LIN {X 0,Y 523.95,Z 318.842,A -85,B 0,C 180,E1 -4818.689,E2 -4818.689} C_VEL
LIN {X 0,Y 523.908,Z 318.846,A -85,B 0,C 180,E1 -4821.08,E2 -4821.08} C_VEL
LIN {X 0,Y 523.913,Z 318.849,A -85,B 0,C 180,E1 -4823.826,E2 -4823.826} C_VEL
LIN {X 0,Y 523.931,Z 318.844,A -85,B 0,C 180,E1 -4826.635,E2 -4826.635} C_VEL
LIN {X 0,Y 523.944,Z 318.837,A -85,B 0,C 180,E1 -4829.355,E2 -4829.355} C_VEL
LIN {X 0,Y 523.929,Z 318.846,A -85,B 0,C 180,E1 -4832.289,E2 -4832.289} C_VEL
LIN {X 0,Y 523.909,Z 318.846,A -85,B 0,C 180,E1 -4835.427,E2 -4835.427} C_VEL
LIN {X 0,Y 523.932,Z 318.841,A -85,B 0,C 180,E1 -4838.766,E2 -4838.766} C_VEL
LIN {X 0,Y 523.923,Z 318.845,A -85,B 0,C 180,E1 -4841.22,E2 -4841.22} C_VEL
LIN {X 0,Y 523.907,Z 318.851,A -85,B 0,C 180,E1 -4843.638,E2 -4843.638} C_VEL
LIN {X 0,Y 523.909,Z 318.849,A -85,B 0,C 180,E1 -4846.027,E2 -4846.027} C_VEL
LIN {X 0,Y 523.947,Z 318.838,A -85,B 0,C 180,E1 -4848.393,E2 -4848.393} C_VEL
LIN {X 0,Y 523.93,Z 318.85,A -85,B 0,C 180,E1 -4851.515,E2 -4851.515} C_VEL
LIN {X 0,Y 524.049,Z 318.827,A -85,B 0,C 180,E1 -4854.614,E2 -4854.614} C_VEL
LIN {X 0,Y 524.086,Z 318.826,A -85,B 0,C 180,E1 -4857.695,E2 -4857.695} C_VEL
LIN {X 0,Y 524.076,Z 318.826,A -85,B 0,C 180,E1 -4860,E2 -4860} C_VEL
LIN {X 0,Y 524.024,Z 318.834,A -85,B 0,C 180,E1 -4863.075,E2 -4863.075} C_VEL
LIN {X 0,Y 524.002,Z 318.833,A -85,B 0,C 180,E1 -4866.16,E2 -4866.16} C_VEL
LIN {X 0,Y 523.966,Z 318.846,A -85,B 0,C 180,E1 -4869.263,E2 -4869.263} C_VEL
LIN {X 0,Y 523.984,Z 318.834,A -85,B 0,C 180,E1 -4871.736,E2 -4871.736} C_VEL
LIN {X 0,Y 523.979,Z 318.844,A -85,B 0,C 180,E1 -4875.052,E2 -4875.052} C_VEL
LIN {X 0,Y 523.935,Z 318.841,A -85,B 0,C 180,E1 -4877.97,E2 -4877.97} C_VEL
LIN {X 0,Y 523.96,Z 318.839,A -85,B 0,C 180,E1 -4880.411,E2 -4880.411} C_VEL
LIN {X 0,Y 523.9,Z 318.855,A -85,B 0,C 180,E1 -4882.894,E2 -4882.894} C_VEL
LIN {X 0,Y 523.942,Z 318.843,A -85,B 0,C 180,E1 -4885.42,E2 -4885.42} C_VEL
LIN {X 0,Y 523.956,Z 318.838,A -85,B 0,C 180,E1 -4888,E2 -4888} C_VEL
LIN {X 0,Y 523.936,Z 318.847,A -85,B 0,C 180,E1 -4890.856,E2 -4890.856} C_VEL
LIN {X 0,Y 523.953,Z 318.839,A -85,B 0,C 180,E1 -4893.736,E2 -4893.736} C_VEL
LIN {X 0,Y 523.897,Z 318.852,A -85,B 0,C 180,E1 -4896.402,E2 -4896.402} C_VEL
LIN {X 0,Y 523.917,Z 318.846,A -85,B 0,C 180,E1 -4899.086,E2 -4899.086} C_VEL
LIN {X 0,Y 523.948,Z 318.844,A -85,B 0,C 180,E1 -4902.12,E2 -4902.12} C_VEL
LIN {X 0,Y 523.95,Z 318.841,A -85,B 0,C 180,E1 -4905.31,E2 -4905.31} C_VEL
LIN {X 0,Y 523.912,Z 318.848,A -85,B 0,C 180,E1 -4906.88,E2 -4906.88} C_VEL
LIN {X 0,Y 523.238,Z 318.931,A -85,B 0,C 180,E1 -4907.522,E2 -4907.522} C_VEL
LIN {X 0,Y 520.371,Z 319.293,A -85,B 0,C 180,E1 -4908.563,E2 -4908.563} C_VEL
LIN {X 0,Y 517.964,Z 319.59,A -85,B 0,C 180,E1 -4909.402,E2 -4909.402} C_VEL
LIN {X 0,Y 516.952,Z 319.717,A -85,B 0,C 180,E1 -4910.05,E2 -4910.05} C_VEL
LIN {X 0,Y 516.88,Z 319.728,A -85,B 0,C 180,E1 -4910.269,E2 -4910.269} C_VEL
LIN {X 0,Y 516.883,Z 319.721,A -85,B 0,C 180,E1 -4913.343,E2 -4913.343} C_VEL
LIN {X 0,Y 516.912,Z 319.723,A -85,B 0,C 180,E1 -4916.122,E2 -4916.122} C_VEL
LIN {X 0,Y 516.892,Z 319.723,A -85,B 0,C 180,E1 -4918.937,E2 -4918.937} C_VEL
LIN {X 0,Y 516.979,Z 319.878,A -85,B 0,C 180,E1 -4921.229,E2 -4921.229} C_VEL
LIN {X 0,Y 518.392,Z 328.272,A -85,B 0,C 180,E1 -4922.771,E2 -4922.771} C_VEL
LIN {X 0,Y 517.957,Z 343.74,A -85,B 0,C 180,E1 -4925.421,E2 -4925.421} C_VEL
LIN {X 0,Y 520.45,Z 355.889,A -85,B 0,C 180,E1 -4925.7,E2 -4925.7} C_VEL
LIN {X 0,Y 519.688,Z 480.334,A -85,B 0,C 180,E1 -4927.462,E2 -4927.462} C_VEL
LIN {X 0,Y 519.494,Z 494.514,A -85,B 0,C 180,E1 -4927.82,E2 -4927.82} C_VEL
LIN {X 0,Y 519.162,Z 507.735,A -85,B 0,C 180,E1 -4928.301,E2 -4928.301} C_VEL
LIN {X 0,Y 518.827,Z 519.994,A -85,B 0,C 180,E1 -4928.891,E2 -4928.891} C_VEL
LIN {X 0,Y 518.403,Z 532.763,A -85,B 0,C 180,E1 -4929.672,E2 -4929.672} C_VEL
LIN {X 0,Y 517.994,Z 544.752,A -85,B 0,C 180,E1 -4930.586,E2 -4930.586} C_VEL
LIN {X 0,Y 517.618,Z 555.659,A -85,B 0,C 180,E1 -4931.599,E2 -4931.599} C_VEL
LIN {X 0,Y 517.261,Z 564.741,A -85,B 0,C 180,E1 -4932.608,E2 -4932.608} C_VEL
LIN {X 0,Y 516.954,Z 573.83,A -85,B 0,C 180,E1 -4933.818,E2 -4933.818} C_VEL
LIN {X 0,Y 516.721,Z 581.347,A -85,B 0,C 180,E1 -4935.024,E2 -4935.024} C_VEL
LIN {X 0,Y 516.572,Z 587.573,A -85,B 0,C 180,E1 -4936.227,E2 -4936.227} C_VEL
LIN {X 0,Y 516.394,Z 592.697,A -85,B 0,C 180,E1 -4937.423,E2 -4937.423} C_VEL
LIN {X 0,Y 516.349,Z 597.948,A -85,B 0,C 180,E1 -4939.015,E2 -4939.015} C_VEL
LIN {X 0,Y 516.193,Z 601.647,A -85,B 0,C 180,E1 -4940.597,E2 -4940.597} C_VEL
LIN {X 0,Y 516.229,Z 603.917,A -85,B 0,C 180,E1 -4942.176,E2 -4942.176} C_VEL
LIN {X 0,Y 516.297,Z 604.832,A -85,B 0,C 180,E1 -4943.748,E2 -4943.748} C_VEL
LIN {X 0,Y 516.214,Z 604.426,A -85,B 0,C 180,E1 -4945.315,E2 -4945.315} C_VEL
LIN {X 0,Y 516.273,Z 602.695,A -85,B 0,C 180,E1 -4946.879,E2 -4946.879} C_VEL
LIN {X 0,Y 516.21,Z 599.622,A -85,B 0,C 180,E1 -4948.44,E2 -4948.44} C_VEL
LIN {X 0,Y 516.286,Z 595.104,A -85,B 0,C 180,E1 -4950,E2 -4950} C_VEL
LIN {X 0,Y 516.389,Z 588.969,A -85,B 0,C 180,E1 -4951.56,E2 -4951.56} C_VEL
LIN {X 0,Y 516.674,Z 582.141,A -85,B 0,C 180,E1 -4952.924,E2 -4952.924} C_VEL
LIN {X 0,Y 516.926,Z 573.712,A -85,B 0,C 180,E1 -4954.288,E2 -4954.288} C_VEL
LIN {X 0,Y 517.277,Z 564.923,A -85,B 0,C 180,E1 -4955.457,E2 -4955.457} C_VEL
LIN {X 0,Y 517.665,Z 554.313,A -85,B 0,C 180,E1 -4956.626,E2 -4956.626} C_VEL
LIN {X 0,Y 518.044,Z 542.812,A -85,B 0,C 180,E1 -4957.667,E2 -4957.667} C_VEL
LIN {X 0,Y 518.539,Z 530.43,A -85,B 0,C 180,E1 -4958.574,E2 -4958.574} C_VEL
LIN {X 0,Y 518.93,Z 517.026,A -85,B 0,C 180,E1 -4959.353,E2 -4959.353} C_VEL
LIN {X 0,Y 519.286,Z 504.042,A -85,B 0,C 180,E1 -4959.936,E2 -4959.936} C_VEL
LIN {X 0,Y 519.641,Z 490.877,A -85,B 0,C 180,E1 -4960.372,E2 -4960.372} C_VEL
LIN {X 0,Y 519.764,Z 476.594,A -85,B 0,C 180,E1 -4960.69,E2 -4960.69} C_VEL
LIN {X 0,Y 520.359,Z 355.201,A -85,B 0,C 180,E1 -4962.402,E2 -4962.402} C_VEL
LIN {X 0,Y 517.922,Z 343.676,A -85,B 0,C 180,E1 -4962.676,E2 -4962.676} C_VEL
LIN {X 0,Y 518.392,Z 328.422,A -85,B 0,C 180,E1 -4965.286,E2 -4965.286} C_VEL
LIN {X 0,Y 517.492,Z 322.48,A -85,B 0,C 180,E1 -4966.367,E2 -4966.367} C_VEL
LIN {X 0,Y 516.924,Z 319.72,A -85,B 0,C 180,E1 -4966.894,E2 -4966.894} C_VEL
LIN {X 0,Y 516.936,Z 319.724,A -85,B 0,C 180,E1 -4969.869,E2 -4969.869} C_VEL
LIN {X 0,Y 516.87,Z 319.725,A -85,B 0,C 180,E1 -4972.389,E2 -4972.389} C_VEL
LIN {X 0,Y 516.878,Z 319.722,A -85,B 0,C 180,E1 -4974.929,E2 -4974.929} C_VEL
LIN {X 0,Y 516.929,Z 319.721,A -85,B 0,C 180,E1 -4977.532,E2 -4977.532} C_VEL
LIN {X 0,Y 516.893,Z 319.722,A -85,B 0,C 180,E1 -4980.203,E2 -4980.203} C_VEL
LIN {X 0,Y 516.897,Z 319.719,A -85,B 0,C 180,E1 -4982.946,E2 -4982.946} C_VEL
LIN {X 0,Y 516.888,Z 319.725,A -85,B 0,C 180,E1 -4985.778,E2 -4985.778} C_VEL
LIN {X 0,Y 516.88,Z 319.721,A -85,B 0,C 180,E1 -4988.715,E2 -4988.715} C_VEL
LIN {X 0,Y 516.908,Z 319.721,A -85,B 0,C 180,E1 -4991.774,E2 -4991.774} C_VEL
LIN {X 0,Y 516.919,Z 319.718,A -85,B 0,C 180,E1 -4995.009,E2 -4995.009} C_VEL
LIN {X 0,Y 516.908,Z 319.715,A -85,B 0,C 180,E1 -4998.398,E2 -4998.398} C_VEL
LIN {X 0,Y 516.874,Z 319.729,A -85,B 0,C 180,E1 -5001.283,E2 -5001.283} C_VEL
LIN {X 0,Y 516.865,Z 319.722,A -85,B 0,C 180,E1 -5004.219,E2 -5004.219} C_VEL
LIN {X 0,Y 516.873,Z 319.726,A -85,B 0,C 180,E1 -5007.051,E2 -5007.051} C_VEL
LIN {X 0,Y 516.882,Z 319.721,A -85,B 0,C 180,E1 -5009.795,E2 -5009.795} C_VEL
LIN {X 0,Y 516.914,Z 319.713,A -85,B 0,C 180,E1 -5012.466,E2 -5012.466} C_VEL
LIN {X 0,Y 516.845,Z 319.733,A -85,B 0,C 180,E1 -5015.068,E2 -5015.068} C_VEL
LIN {X 0,Y 516.858,Z 319.722,A -85,B 0,C 180,E1 -5017.621,E2 -5017.621} C_VEL
LIN {X 0,Y 516.917,Z 319.71,A -85,B 0,C 180,E1 -5020.129,E2 -5020.129} C_VEL
LIN {X 0,Y 516.883,Z 319.723,A -85,B 0,C 180,E1 -5022.594,E2 -5022.594} C_VEL
LIN {X 0,Y 516.927,Z 319.718,A -85,B 0,C 180,E1 -5025.029,E2 -5025.029} C_VEL
LIN {X 0,Y 516.953,Z 319.707,A -85,B 0,C 180,E1 -5028.233,E2 -5028.233} C_VEL
LIN {X 0,Y 516.937,Z 319.714,A -85,B 0,C 180,E1 -5031.399,E2 -5031.399} C_VEL
LIN {X 0,Y 516.969,Z 319.707,A -85,B 0,C 180,E1 -5033.756,E2 -5033.756} C_VEL
LIN {X 0,Y 516.964,Z 319.713,A -85,B 0,C 180,E1 -5036.882,E2 -5036.882} C_VEL
LIN {X 0,Y 516.95,Z 319.717,A -85,B 0,C 180,E1 -5038.442,E2 -5038.442} C_VEL
LIN {X 0,Y 517.075,Z 319.7,A -85,B 0,C 180,E1 -5040.779,E2 -5040.779} C_VEL
LIN {X 0,Y 516.927,Z 319.712,A -85,B 0,C 180,E1 -5043.117,E2 -5043.117} C_VEL
LIN {X 0,Y 516.955,Z 319.717,A -85,B 0,C 180,E1 -5046.244,E2 -5046.244} C_VEL
LIN {X 0,Y 516.918,Z 319.711,A -85,B 0,C 180,E1 -5049.39,E2 -5049.39} C_VEL
LIN {X 0,Y 516.938,Z 319.715,A -85,B 0,C 180,E1 -5051.807,E2 -5051.807} C_VEL
LIN {X 0,Y 516.931,Z 319.711,A -85,B 0,C 180,E1 -5055.146,E2 -5055.146} C_VEL
LIN {X 0,Y 516.898,Z 319.727,A -85,B 0,C 180,E1 -5058.223,E2 -5058.223} C_VEL
LIN {X 0,Y 516.892,Z 319.717,A -85,B 0,C 180,E1 -5060.702,E2 -5060.702} C_VEL
LIN {X 0,Y 516.877,Z 319.729,A -85,B 0,C 180,E1 -5064.074,E2 -5064.074} C_VEL
LIN {X 0,Y 516.884,Z 319.72,A -85,B 0,C 180,E1 -5066.66,E2 -5066.66} C_VEL
LIN {X 0,Y 516.898,Z 319.72,A -85,B 0,C 180,E1 -5069.524,E2 -5069.524} C_VEL
LIN {X 0,Y 516.885,Z 319.721,A -85,B 0,C 180,E1 -5072.544,E2 -5072.544} C_VEL
LIN {X 0,Y 516.866,Z 319.724,A -85,B 0,C 180,E1 -5075.332,E2 -5075.332} C_VEL
LIN {X 0,Y 516.871,Z 319.729,A -85,B 0,C 180,E1 -5077.944,E2 -5077.944} C_VEL
LIN {X 0,Y 516.876,Z 319.718,A -85,B 0,C 180,E1 -5080.742,E2 -5080.742} C_VEL
LIN {X 0,Y 516.875,Z 319.72,A -85,B 0,C 180,E1 -5082.832,E2 -5082.832} C_VEL
LIN {X 0,Y 516.916,Z 319.717,A -85,B 0,C 180,E1 -5085.011,E2 -5085.011} C_VEL
LIN {X 0,Y 516.909,Z 319.718,A -85,B 0,C 180,E1 -5088.399,E2 -5088.399} C_VEL
LIN {X 0,Y 516.875,Z 319.728,A -85,B 0,C 180,E1 -5091.285,E2 -5091.285} C_VEL
LIN {X 0,Y 516.884,Z 319.723,A -85,B 0,C 180,E1 -5094.222,E2 -5094.222} C_VEL
LIN {X 0,Y 516.892,Z 319.724,A -85,B 0,C 180,E1 -5097.054,E2 -5097.054} C_VEL
LIN {X 0,Y 516.889,Z 319.724,A -85,B 0,C 180,E1 -5099.797,E2 -5099.797} C_VEL
LIN {X 0,Y 516.924,Z 319.718,A -85,B 0,C 180,E1 -5102.468,E2 -5102.468} C_VEL
LIN {X 0,Y 516.958,Z 319.835,A -85,B 0,C 180,E1 -5103.831,E2 -5103.831} C_VEL
LIN {X 0,Y 519.186,Z 331.01,A -85,B 0,C 180,E1 -5105.616,E2 -5105.616} C_VEL
LIN {X 0,Y 518.581,Z 350.946,A -85,B 0,C 180,E1 -5108.537,E2 -5108.537} C_VEL
LIN {X 0,Y 517.999,Z 370.569,A -85,B 0,C 180,E1 -5111.367,E2 -5111.367} C_VEL
LIN {X 0,Y 520.414,Z 384.995,A -85,B 0,C 180,E1 -5111.669,E2 -5111.669} C_VEL
LIN {X 0,Y 519.633,Z 509.029,A -85,B 0,C 180,E1 -5113.424,E2 -5113.424} C_VEL
LIN {X 0,Y 519.37,Z 523.154,A -85,B 0,C 180,E1 -5113.781,E2 -5113.781} C_VEL
LIN {X 0,Y 519.054,Z 536.913,A -85,B 0,C 180,E1 -5114.289,E2 -5114.289} C_VEL
LIN {X 0,Y 518.638,Z 550.885,A -85,B 0,C 180,E1 -5114.98,E2 -5114.98} C_VEL
LIN {X 0,Y 518.213,Z 563.388,A -85,B 0,C 180,E1 -5115.771,E2 -5115.771} C_VEL
LIN {X 0,Y 517.75,Z 575.993,A -85,B 0,C 180,E1 -5116.758,E2 -5116.758} C_VEL
LIN {X 0,Y 517.401,Z 587.135,A -85,B 0,C 180,E1 -5117.836,E2 -5117.836} C_VEL
LIN {X 0,Y 517.093,Z 597.302,A -85,B 0,C 180,E1 -5119.031,E2 -5119.031} C_VEL
LIN {X 0,Y 516.779,Z 605.67,A -85,B 0,C 180,E1 -5120.213,E2 -5120.213} C_VEL
LIN {X 0,Y 516.582,Z 613.673,A -85,B 0,C 180,E1 -5121.59,E2 -5121.59} C_VEL
LIN {X 0,Y 516.401,Z 620.117,A -85,B 0,C 180,E1 -5122.965,E2 -5122.965} C_VEL
LIN {X 0,Y 516.407,Z 624.584,A -85,B 0,C 180,E1 -5124.142,E2 -5124.142} C_VEL
LIN {X 0,Y 516.264,Z 628.09,A -85,B 0,C 180,E1 -5125.315,E2 -5125.315} C_VEL
LIN {X 0,Y 516.324,Z 629.979,A -85,B 0,C 180,E1 -5126.098,E2 -5126.098} C_VEL
LIN {X 0,Y 516.259,Z 632.685,A -85,B 0,C 180,E1 -5127.659,E2 -5127.659} C_VEL
LIN {X 0,Y 516.157,Z 634.024,A -85,B 0,C 180,E1 -5129.22,E2 -5129.22} C_VEL
LIN {X 0,Y 516.157,Z 634.024,A -85,B 0,C 180,E1 -5130.78,E2 -5130.78} C_VEL
LIN {X 0,Y 516.259,Z 632.686,A -85,B 0,C 180,E1 -5132.341,E2 -5132.341} C_VEL
LIN {X 0,Y 516.324,Z 629.98,A -85,B 0,C 180,E1 -5133.902,E2 -5133.902} C_VEL
LIN {X 0,Y 516.367,Z 625.828,A -85,B 0,C 180,E1 -5135.467,E2 -5135.467} C_VEL
LIN {X 0,Y 516.401,Z 620.109,A -85,B 0,C 180,E1 -5137.035,E2 -5137.035} C_VEL
LIN {X 0,Y 516.582,Z 613.665,A -85,B 0,C 180,E1 -5138.41,E2 -5138.41} C_VEL
LIN {X 0,Y 516.778,Z 605.659,A -85,B 0,C 180,E1 -5139.787,E2 -5139.787} C_VEL
LIN {X 0,Y 517.078,Z 597.289,A -85,B 0,C 180,E1 -5140.969,E2 -5140.969} C_VEL
LIN {X 0,Y 517.413,Z 586.881,A -85,B 0,C 180,E1 -5142.19,E2 -5142.19} C_VEL
LIN {X 0,Y 517.782,Z 575.975,A -85,B 0,C 180,E1 -5143.241,E2 -5143.241} C_VEL
LIN {X 0,Y 518.21,Z 563.371,A -85,B 0,C 180,E1 -5144.229,E2 -5144.229} C_VEL
LIN {X 0,Y 518.658,Z 550.865,A -85,B 0,C 180,E1 -5145.019,E2 -5145.019} C_VEL
LIN {X 0,Y 519.055,Z 538.011,A -85,B 0,C 180,E1 -5145.661,E2 -5145.661} C_VEL
LIN {X 0,Y 519.318,Z 524.346,A -85,B 0,C 180,E1 -5146.18,E2 -5146.18} C_VEL
LIN {X 0,Y 519.612,Z 510.139,A -85,B 0,C 180,E1 -5146.551,E2 -5146.551} C_VEL
LIN {X 0,Y 519.846,Z 482.014,A -85,B 0,C 180,E1 -5146.973,E2 -5146.973} C_VEL
LIN {X 0,Y 520.349,Z 384.013,A -85,B 0,C 180,E1 -5148.347,E2 -5148.347} C_VEL
LIN {X 0,Y 518,Z 370.517,A -85,B 0,C 180,E1 -5148.636,E2 -5148.636} C_VEL
LIN {X 0,Y 518.599,Z 349.484,A -85,B 0,C 180,E1 -5151.671,E2 -5151.671} C_VEL
LIN {X 0,Y 519.182,Z 330.987,A -85,B 0,C 180,E1 -5154.384,E2 -5154.384} C_VEL
LIN {X 0,Y 516.941,Z 319.775,A -85,B 0,C 180,E1 -5156.195,E2 -5156.195} C_VEL
LIN {X 0,Y 516.919,Z 319.719,A -85,B 0,C 180,E1 -5159.304,E2 -5159.304} C_VEL
LIN {X 0,Y 516.892,Z 319.728,A -85,B 0,C 180,E1 -5162.543,E2 -5162.543} C_VEL
LIN {X 0,Y 516.875,Z 319.722,A -85,B 0,C 180,E1 -5165.331,E2 -5165.331} C_VEL
LIN {X 0,Y 516.876,Z 319.72,A -85,B 0,C 180,E1 -5167.942,E2 -5167.942} C_VEL
LIN {X 0,Y 516.878,Z 319.722,A -85,B 0,C 180,E1 -5170.741,E2 -5170.741} C_VEL
LIN {X 0,Y 516.876,Z 319.721,A -85,B 0,C 180,E1 -5172.831,E2 -5172.831} C_VEL
LIN {X 0,Y 516.916,Z 319.714,A -85,B 0,C 180,E1 -5175.009,E2 -5175.009} C_VEL
LIN {X 0,Y 516.907,Z 319.723,A -85,B 0,C 180,E1 -5178.398,E2 -5178.398} C_VEL
LIN {X 0,Y 516.871,Z 319.722,A -85,B 0,C 180,E1 -5181.283,E2 -5181.283} C_VEL
LIN {X 0,Y 516.876,Z 319.727,A -85,B 0,C 180,E1 -5184.22,E2 -5184.22} C_VEL
LIN {X 0,Y 516.884,Z 319.72,A -85,B 0,C 180,E1 -5187.052,E2 -5187.052} C_VEL
LIN {X 0,Y 516.88,Z 319.719,A -85,B 0,C 180,E1 -5189.796,E2 -5189.796} C_VEL
LIN {X 0,Y 516.881,Z 319.722,A -85,B 0,C 180,E1 -5192.465,E2 -5192.465} C_VEL
LIN {X 0,Y 516.853,Z 319.723,A -85,B 0,C 180,E1 -5195.069,E2 -5195.069} C_VEL
LIN {X 0,Y 516.856,Z 319.729,A -85,B 0,C 180,E1 -5197.621,E2 -5197.621} C_VEL
LIN {X 0,Y 516.916,Z 319.72,A -85,B 0,C 180,E1 -5200.129,E2 -5200.129} C_VEL
LIN {X 0,Y 516.881,Z 319.72,A -85,B 0,C 180,E1 -5202.595,E2 -5202.595} C_VEL
LIN {X 0,Y 516.921,Z 319.715,A -85,B 0,C 180,E1 -5205.03,E2 -5205.03} C_VEL
LIN {X 0,Y 516.911,Z 319.715,A -85,B 0,C 180,E1 -5208.233,E2 -5208.233} C_VEL
LIN {X 0,Y 516.904,Z 319.725,A -85,B 0,C 180,E1 -5211.399,E2 -5211.399} C_VEL
LIN {X 0,Y 516.995,Z 319.706,A -85,B 0,C 180,E1 -5214.54,E2 -5214.54} C_VEL
LIN {X 0,Y 517.058,Z 319.701,A -85,B 0,C 180,E1 -5217.663,E2 -5217.663} C_VEL
LIN {X 0,Y 517.045,Z 319.701,A -85,B 0,C 180,E1 -5220,E2 -5220} C_VEL
LIN {X 0,Y 517.059,Z 319.696,A -85,B 0,C 180,E1 -5222.337,E2 -5222.337} C_VEL
LIN {X 0,Y 517,Z 319.711,A -85,B 0,C 180,E1 -5225.461,E2 -5225.461} C_VEL
LIN {X 0,Y 516.948,Z 319.712,A -85,B 0,C 180,E1 -5227.814,E2 -5227.814} C_VEL
LIN {X 0,Y 516.931,Z 319.721,A -85,B 0,C 180,E1 -5230.973,E2 -5230.973} C_VEL
LIN {X 0,Y 516.872,Z 319.722,A -85,B 0,C 180,E1 -5234.167,E2 -5234.167} C_VEL
LIN {X 0,Y 516.894,Z 319.72,A -85,B 0,C 180,E1 -5236.591,E2 -5236.591} C_VEL
LIN {X 0,Y 516.888,Z 319.727,A -85,B 0,C 180,E1 -5239.046,E2 -5239.046} C_VEL
LIN {X 0,Y 516.874,Z 319.723,A -85,B 0,C 180,E1 -5241.539,E2 -5241.539} C_VEL
LIN {X 0,Y 516.898,Z 319.725,A -85,B 0,C 180,E1 -5244.929,E2 -5244.929} C_VEL
LIN {X 0,Y 516.913,Z 319.715,A -85,B 0,C 180,E1 -5247.906,E2 -5247.906} C_VEL
LIN {X 0,Y 516.883,Z 319.722,A -85,B 0,C 180,E1 -5250.205,E2 -5250.205} C_VEL
LIN {X 0,Y 516.889,Z 319.724,A -85,B 0,C 180,E1 -5252.948,E2 -5252.948} C_VEL
LIN {X 0,Y 516.865,Z 319.722,A -85,B 0,C 180,E1 -5255.781,E2 -5255.781} C_VEL
LIN {X 0,Y 516.876,Z 319.727,A -85,B 0,C 180,E1 -5258.717,E2 -5258.717} C_VEL
LIN {X 0,Y 516.909,Z 319.718,A -85,B 0,C 180,E1 -5261.776,E2 -5261.776} C_VEL
LIN {X 0,Y 516.919,Z 319.718,A -85,B 0,C 180,E1 -5265.011,E2 -5265.011} C_VEL
LIN {X 0,Y 516.912,Z 319.724,A -85,B 0,C 180,E1 -5268.4,E2 -5268.4} C_VEL
LIN {X 0,Y 516.88,Z 319.728,A -85,B 0,C 180,E1 -5270.269,E2 -5270.269} C_VEL
LIN {X 0,Y 516.244,Z 319.814,A -85,B 0,C 180,E1 -5270.919,E2 -5270.919} C_VEL
LIN {X 0,Y 513.402,Z 320.167,A -85,B 0,C 180,E1 -5271.974,E2 -5271.974} C_VEL
LIN {X 0,Y 510.975,Z 320.463,A -85,B 0,C 180,E1 -5272.824,E2 -5272.824} C_VEL
LIN {X 0,Y 509.921,Z 320.59,A -85,B 0,C 180,E1 -5273.481,E2 -5273.481} C_VEL
LIN {X 0,Y 509.831,Z 320.601,A -85,B 0,C 180,E1 -5273.703,E2 -5273.703} C_VEL
LIN {X 0,Y 509.862,Z 320.601,A -85,B 0,C 180,E1 -5276.54,E2 -5276.54} C_VEL
LIN {X 0,Y 509.847,Z 320.601,A -85,B 0,C 180,E1 -5279.335,E2 -5279.335} C_VEL
LIN {X 0,Y 509.901,Z 320.629,A -85,B 0,C 180,E1 -5280.989,E2 -5280.989} C_VEL
LIN {X 0,Y 511.449,Z 329.163,A -85,B 0,C 180,E1 -5282.592,E2 -5282.592} C_VEL
LIN {X 0,Y 511.05,Z 343.771,A -85,B 0,C 180,E1 -5285.132,E2 -5285.132} C_VEL
LIN {X 0,Y 511.206,Z 344.967,A -85,B 0,C 180,E1 -5285.193,E2 -5285.193} C_VEL
LIN {X 0,Y 513.725,Z 357.045,A -85,B 0,C 180,E1 -5285.465,E2 -5285.465} C_VEL
LIN {X 0,Y 512.908,Z 480.339,A -85,B 0,C 180,E1 -5287.233,E2 -5287.233} C_VEL
LIN {X 0,Y 512.696,Z 494.434,A -85,B 0,C 180,E1 -5287.589,E2 -5287.589} C_VEL
LIN {X 0,Y 512.328,Z 508.308,A -85,B 0,C 180,E1 -5288.103,E2 -5288.103} C_VEL
LIN {X 0,Y 511.96,Z 520.665,A -85,B 0,C 180,E1 -5288.71,E2 -5288.71} C_VEL
LIN {X 0,Y 511.514,Z 533.228,A -85,B 0,C 180,E1 -5289.494,E2 -5289.494} C_VEL
LIN {X 0,Y 511.065,Z 545.144,A -85,B 0,C 180,E1 -5290.416,E2 -5290.416} C_VEL
LIN {X 0,Y 510.718,Z 555.025,A -85,B 0,C 180,E1 -5291.341,E2 -5291.341} C_VEL
LIN {X 0,Y 510.313,Z 564.247,A -85,B 0,C 180,E1 -5292.364,E2 -5292.364} C_VEL
LIN {X 0,Y 509.937,Z 573.452,A -85,B 0,C 180,E1 -5293.589,E2 -5293.589} C_VEL
LIN {X 0,Y 509.679,Z 581.963,A -85,B 0,C 180,E1 -5294.973,E2 -5294.973} C_VEL
LIN {X 0,Y 509.446,Z 589.219,A -85,B 0,C 180,E1 -5296.437,E2 -5296.437} C_VEL
LIN {X 0,Y 509.314,Z 594.04,A -85,B 0,C 180,E1 -5297.65,E2 -5297.65} C_VEL
LIN {X 0,Y 509.226,Z 598.997,A -85,B 0,C 180,E1 -5299.262,E2 -5299.262} C_VEL
LIN {X 0,Y 509.108,Z 601.696,A -85,B 0,C 180,E1 -5300.465,E2 -5300.465} C_VEL
LIN {X 0,Y 509.143,Z 604.035,A -85,B 0,C 180,E1 -5302.066,E2 -5302.066} C_VEL
LIN {X 0,Y 509.223,Z 605.016,A -85,B 0,C 180,E1 -5303.661,E2 -5303.661} C_VEL
LIN {X 0,Y 509.13,Z 604.677,A -85,B 0,C 180,E1 -5305.249,E2 -5305.249} C_VEL
LIN {X 0,Y 509.189,Z 603.012,A -85,B 0,C 180,E1 -5306.835,E2 -5306.835} C_VEL
LIN {X 0,Y 509.129,Z 600.008,A -85,B 0,C 180,E1 -5308.418,E2 -5308.418} C_VEL
LIN {X 0,Y 509.203,Z 595.577,A -85,B 0,C 180,E1 -5310,E2 -5310} C_VEL
LIN {X 0,Y 509.359,Z 591.183,A -85,B 0,C 180,E1 -5311.186,E2 -5311.186} C_VEL
LIN {X 0,Y 509.402,Z 585.867,A -85,B 0,C 180,E1 -5312.372,E2 -5312.372} C_VEL
LIN {X 0,Y 509.809,Z 578.244,A -85,B 0,C 180,E1 -5313.754,E2 -5313.754} C_VEL
LIN {X 0,Y 510.036,Z 570.335,A -85,B 0,C 180,E1 -5314.94,E2 -5314.94} C_VEL
LIN {X 0,Y 510.472,Z 560.809,A -85,B 0,C 180,E1 -5316.125,E2 -5316.125} C_VEL
LIN {X 0,Y 510.846,Z 551.329,A -85,B 0,C 180,E1 -5317.112,E2 -5317.112} C_VEL
LIN {X 0,Y 511.261,Z 539.04,A -85,B 0,C 180,E1 -5318.169,E2 -5318.169} C_VEL
LIN {X 0,Y 511.764,Z 527.273,A -85,B 0,C 180,E1 -5318.987,E2 -5318.987} C_VEL
LIN {X 0,Y 512.184,Z 514.945,A -85,B 0,C 180,E1 -5319.676,E2 -5319.676} C_VEL
LIN {X 0,Y 512.523,Z 501.271,A -85,B 0,C 180,E1 -5320.268,E2 -5320.268} C_VEL
LIN {X 0,Y 512.864,Z 486.886,A -85,B 0,C 180,E1 -5320.711,E2 -5320.711} C_VEL
LIN {X 0,Y 513.026,Z 472.695,A -85,B 0,C 180,E1 -5320.982,E2 -5320.982} C_VEL
LIN {X 0,Y 513.669,Z 356.374,A -85,B 0,C 180,E1 -5322.636,E2 -5322.636} C_VEL
LIN {X 0,Y 511.017,Z 343.888,A -85,B 0,C 180,E1 -5322.934,E2 -5322.934} C_VEL
LIN {X 0,Y 511.469,Z 329.787,A -85,B 0,C 180,E1 -5325.376,E2 -5325.376} C_VEL
LIN {X 0,Y 510.169,Z 322.01,A -85,B 0,C 180,E1 -5326.815,E2 -5326.815} C_VEL
LIN {X 0,Y 509.898,Z 320.596,A -85,B 0,C 180,E1 -5327.082,E2 -5327.082} C_VEL
LIN {X 0,Y 509.89,Z 320.597,A -85,B 0,C 180,E1 -5330.401,E2 -5330.401} C_VEL
LIN {X 0,Y 509.825,Z 320.605,A -85,B 0,C 180,E1 -5333.563,E2 -5333.563} C_VEL
LIN {X 0,Y 509.914,Z 320.591,A -85,B 0,C 180,E1 -5336.378,E2 -5336.378} C_VEL
LIN {X 0,Y 509.877,Z 320.592,A -85,B 0,C 180,E1 -5338.843,E2 -5338.843} C_VEL
LIN {X 0,Y 509.823,Z 320.607,A -85,B 0,C 180,E1 -5341.589,E2 -5341.589} C_VEL
LIN {X 0,Y 509.853,Z 320.596,A -85,B 0,C 180,E1 -5344.412,E2 -5344.412} C_VEL
LIN {X 0,Y 509.817,Z 320.605,A -85,B 0,C 180,E1 -5347.339,E2 -5347.339} C_VEL
LIN {X 0,Y 509.835,Z 320.592,A -85,B 0,C 180,E1 -5350.381,E2 -5350.381} C_VEL
LIN {X 0,Y 509.819,Z 320.603,A -85,B 0,C 180,E1 -5353.061,E2 -5353.061} C_VEL
LIN {X 0,Y 509.827,Z 320.603,A -85,B 0,C 180,E1 -5355.791,E2 -5355.791} C_VEL
LIN {X 0,Y 509.85,Z 320.595,A -85,B 0,C 180,E1 -5358.573,E2 -5358.573} C_VEL
LIN {X 0,Y 509.844,Z 320.597,A -85,B 0,C 180,E1 -5361.785,E2 -5361.785} C_VEL
LIN {X 0,Y 509.824,Z 320.601,A -85,B 0,C 180,E1 -5364.621,E2 -5364.621} C_VEL
LIN {X 0,Y 509.851,Z 320.6,A -85,B 0,C 180,E1 -5367.48,E2 -5367.48} C_VEL
LIN {X 0,Y 509.85,Z 320.596,A -85,B 0,C 180,E1 -5370.273,E2 -5370.273} C_VEL
LIN {X 0,Y 509.865,Z 320.596,A -85,B 0,C 180,E1 -5372.943,E2 -5372.943} C_VEL
LIN {X 0,Y 509.83,Z 320.601,A -85,B 0,C 180,E1 -5375.572,E2 -5375.572} C_VEL
LIN {X 0,Y 509.81,Z 320.599,A -85,B 0,C 180,E1 -5378.148,E2 -5378.148} C_VEL
LIN {X 0,Y 509.845,Z 320.596,A -85,B 0,C 180,E1 -5380.68,E2 -5380.68} C_VEL
LIN {X 0,Y 509.852,Z 320.6,A -85,B 0,C 180,E1 -5383.173,E2 -5383.173} C_VEL
LIN {X 0,Y 509.843,Z 320.594,A -85,B 0,C 180,E1 -5385.633,E2 -5385.633} C_VEL
LIN {X 0,Y 509.894,Z 320.595,A -85,B 0,C 180,E1 -5388.874,E2 -5388.874} C_VEL
LIN {X 0,Y 509.906,Z 320.59,A -85,B 0,C 180,E1 -5392.077,E2 -5392.077} C_VEL
LIN {X 0,Y 509.949,Z 320.587,A -85,B 0,C 180,E1 -5394.464,E2 -5394.464} C_VEL
LIN {X 0,Y 510.028,Z 320.572,A -85,B 0,C 180,E1 -5397.631,E2 -5397.631} C_VEL
LIN {X 0,Y 510.024,Z 320.578,A -85,B 0,C 180,E1 -5400.789,E2 -5400.789} C_VEL
LIN {X 0,Y 509.871,Z 320.591,A -85,B 0,C 180,E1 -5403.16,E2 -5403.16} C_VEL
LIN {X 0,Y 509.903,Z 320.597,A -85,B 0,C 180,E1 -5406.33,E2 -5406.33} C_VEL
LIN {X 0,Y 509.858,Z 320.591,A -85,B 0,C 180,E1 -5409.521,E2 -5409.521} C_VEL
LIN {X 0,Y 509.89,Z 320.594,A -85,B 0,C 180,E1 -5411.932,E2 -5411.932} C_VEL
LIN {X 0,Y 509.881,Z 320.589,A -85,B 0,C 180,E1 -5415.242,E2 -5415.242} C_VEL
LIN {X 0,Y 509.843,Z 320.601,A -85,B 0,C 180,E1 -5418.484,E2 -5418.484} C_VEL
LIN {X 0,Y 509.833,Z 320.594,A -85,B 0,C 180,E1 -5421.002,E2 -5421.002} C_VEL
LIN {X 0,Y 509.809,Z 320.602,A -85,B 0,C 180,E1 -5423.564,E2 -5423.564} C_VEL
LIN {X 0,Y 509.866,Z 320.597,A -85,B 0,C 180,E1 -5426.371,E2 -5426.371} C_VEL
LIN {X 0,Y 509.846,Z 320.602,A -85,B 0,C 180,E1 -5429.752,E2 -5429.752} C_VEL
LIN {X 0,Y 509.862,Z 320.595,A -85,B 0,C 180,E1 -5432.775,E2 -5432.775} C_VEL
LIN {X 0,Y 509.827,Z 320.603,A -85,B 0,C 180,E1 -5435.581,E2 -5435.581} C_VEL
LIN {X 0,Y 509.84,Z 320.6,A -85,B 0,C 180,E1 -5438.339,E2 -5438.339} C_VEL
LIN {X 0,Y 509.849,Z 320.598,A -85,B 0,C 180,E1 -5441.426,E2 -5441.426} C_VEL
LIN {X 0,Y 509.85,Z 320.596,A -85,B 0,C 180,E1 -5444.669,E2 -5444.669} C_VEL
LIN {X 0,Y 509.851,Z 320.599,A -85,B 0,C 180,E1 -5448.104,E2 -5448.104} C_VEL
LIN {X 0,Y 509.84,Z 320.599,A -85,B 0,C 180,E1 -5450.648,E2 -5450.648} C_VEL
LIN {X 0,Y 509.83,Z 320.608,A -85,B 0,C 180,E1 -5453.649,E2 -5453.649} C_VEL
LIN {X 0,Y 509.857,Z 320.597,A -85,B 0,C 180,E1 -5456.54,E2 -5456.54} C_VEL
LIN {X 0,Y 509.842,Z 320.605,A -85,B 0,C 180,E1 -5459.335,E2 -5459.335} C_VEL
LIN {X 0,Y 509.89,Z 320.596,A -85,B 0,C 180,E1 -5462.055,E2 -5462.055} C_VEL
LIN {X 0,Y 509.914,Z 320.746,A -85,B 0,C 180,E1 -5463.621,E2 -5463.621} C_VEL
LIN {X 0,Y 512.29,Z 332.48,A -85,B 0,C 180,E1 -5465.521,E2 -5465.521} C_VEL
LIN {X 0,Y 511.646,Z 352.18,A -85,B 0,C 180,E1 -5468.443,E2 -5468.443} C_VEL
LIN {X 0,Y 511.076,Z 370.394,A -85,B 0,C 180,E1 -5471.109,E2 -5471.109} C_VEL
LIN {X 0,Y 513.687,Z 385.81,A -85,B 0,C 180,E1 -5471.435,E2 -5471.435} C_VEL
LIN {X 0,Y 512.817,Z 508.816,A -85,B 0,C 180,E1 -5473.197,E2 -5473.197} C_VEL
LIN {X 0,Y 512.527,Z 523.27,A -85,B 0,C 180,E1 -5473.569,E2 -5473.569} C_VEL
LIN {X 0,Y 512.206,Z 536.706,A -85,B 0,C 180,E1 -5474.073,E2 -5474.073} C_VEL
LIN {X 0,Y 511.771,Z 550.68,A -85,B 0,C 180,E1 -5474.774,E2 -5474.774} C_VEL
LIN {X 0,Y 511.273,Z 563.183,A -85,B 0,C 180,E1 -5475.573,E2 -5475.573} C_VEL
LIN {X 0,Y 510.805,Z 575.789,A -85,B 0,C 180,E1 -5476.575,E2 -5476.575} C_VEL
LIN {X 0,Y 510.409,Z 586.355,A -85,B 0,C 180,E1 -5477.604,E2 -5477.604} C_VEL
LIN {X 0,Y 510.063,Z 597.098,A -85,B 0,C 180,E1 -5478.878,E2 -5478.878} C_VEL
LIN {X 0,Y 509.732,Z 605.467,A -85,B 0,C 180,E1 -5480.076,E2 -5480.076} C_VEL
LIN {X 0,Y 509.522,Z 613.471,A -85,B 0,C 180,E1 -5481.473,E2 -5481.473} C_VEL
LIN {X 0,Y 509.326,Z 619.915,A -85,B 0,C 180,E1 -5482.866,E2 -5482.866} C_VEL
LIN {X 0,Y 509.304,Z 624.382,A -85,B 0,C 180,E1 -5484.06,E2 -5484.06} C_VEL
LIN {X 0,Y 509.181,Z 627.889,A -85,B 0,C 180,E1 -5485.25,E2 -5485.25} C_VEL
LIN {X 0,Y 509.193,Z 631.305,A -85,B 0,C 180,E1 -5486.835,E2 -5486.835} C_VEL
LIN {X 0,Y 509.109,Z 633.322,A -85,B 0,C 180,E1 -5488.418,E2 -5488.418} C_VEL
LIN {X 0,Y 509.064,Z 633.99,A -85,B 0,C 180,E1 -5490,E2 -5490} C_VEL
LIN {X 0,Y 509.109,Z 633.322,A -85,B 0,C 180,E1 -5491.582,E2 -5491.582} C_VEL
LIN {X 0,Y 509.193,Z 631.305,A -85,B 0,C 180,E1 -5493.165,E2 -5493.165} C_VEL
LIN {X 0,Y 509.181,Z 627.886,A -85,B 0,C 180,E1 -5494.75,E2 -5494.75} C_VEL
LIN {X 0,Y 509.303,Z 624.373,A -85,B 0,C 180,E1 -5495.94,E2 -5495.94} C_VEL
LIN {X 0,Y 509.326,Z 619.904,A -85,B 0,C 180,E1 -5497.134,E2 -5497.134} C_VEL
LIN {X 0,Y 509.522,Z 613.46,A -85,B 0,C 180,E1 -5498.527,E2 -5498.527} C_VEL
LIN {X 0,Y 509.731,Z 605.452,A -85,B 0,C 180,E1 -5499.924,E2 -5499.924} C_VEL
LIN {X 0,Y 510.047,Z 597.081,A -85,B 0,C 180,E1 -5501.122,E2 -5501.122} C_VEL
LIN {X 0,Y 510.411,Z 586.364,A -85,B 0,C 180,E1 -5502.393,E2 -5502.393} C_VEL
LIN {X 0,Y 510.819,Z 575.765,A -85,B 0,C 180,E1 -5503.425,E2 -5503.425} C_VEL
LIN {X 0,Y 511.231,Z 564.59,A -85,B 0,C 180,E1 -5504.326,E2 -5504.326} C_VEL
LIN {X 0,Y 511.687,Z 552.424,A -85,B 0,C 180,E1 -5505.127,E2 -5505.127} C_VEL
LIN {X 0,Y 512.167,Z 538.93,A -85,B 0,C 180,E1 -5505.826,E2 -5505.826} C_VEL
LIN {X 0,Y 512.466,Z 524.772,A -85,B 0,C 180,E1 -5506.381,E2 -5506.381} C_VEL
LIN {X 0,Y 512.814,Z 509.919,A -85,B 0,C 180,E1 -5506.777,E2 -5506.777} C_VEL
LIN {X 0,Y 513.028,Z 483.59,A -85,B 0,C 180,E1 -5507.18,E2 -5507.18} C_VEL
LIN {X 0,Y 513.571,Z 384.829,A -85,B 0,C 180,E1 -5508.583,E2 -5508.583} C_VEL
LIN {X 0,Y 511.08,Z 370.329,A -85,B 0,C 180,E1 -5508.895,E2 -5508.895} C_VEL
LIN {X 0,Y 511.698,Z 349.298,A -85,B 0,C 180,E1 -5511.979,E2 -5511.979} C_VEL
LIN {X 0,Y 512.29,Z 332.536,A -85,B 0,C 180,E1 -5514.479,E2 -5514.479} C_VEL
LIN {X 0,Y 510.286,Z 322.35,A -85,B 0,C 180,E1 -5516.149,E2 -5516.149} C_VEL
LIN {X 0,Y 509.905,Z 320.598,A -85,B 0,C 180,E1 -5516.485,E2 -5516.485} C_VEL
LIN {X 0,Y 509.874,Z 320.6,A -85,B 0,C 180,E1 -5518.844,E2 -5518.844} C_VEL
LIN {X 0,Y 509.816,Z 320.603,A -85,B 0,C 180,E1 -5521.589,E2 -5521.589} C_VEL
LIN {X 0,Y 509.848,Z 320.604,A -85,B 0,C 180,E1 -5524.413,E2 -5524.413} C_VEL
LIN {X 0,Y 509.814,Z 320.597,A -85,B 0,C 180,E1 -5527.34,E2 -5527.34} C_VEL
LIN {X 0,Y 509.832,Z 320.6,A -85,B 0,C 180,E1 -5530.381,E2 -5530.381} C_VEL
LIN {X 0,Y 509.816,Z 320.599,A -85,B 0,C 180,E1 -5533.061,E2 -5533.061} C_VEL
LIN {X 0,Y 509.823,Z 320.599,A -85,B 0,C 180,E1 -5535.792,E2 -5535.792} C_VEL
LIN {X 0,Y 509.849,Z 320.6,A -85,B 0,C 180,E1 -5538.574,E2 -5538.574} C_VEL
LIN {X 0,Y 509.842,Z 320.602,A -85,B 0,C 180,E1 -5541.786,E2 -5541.786} C_VEL
LIN {X 0,Y 509.83,Z 320.599,A -85,B 0,C 180,E1 -5544.622,E2 -5544.622} C_VEL
LIN {X 0,Y 509.851,Z 320.598,A -85,B 0,C 180,E1 -5547.48,E2 -5547.48} C_VEL
LIN {X 0,Y 509.847,Z 320.594,A -85,B 0,C 180,E1 -5550.273,E2 -5550.273} C_VEL
LIN {X 0,Y 509.863,Z 320.599,A -85,B 0,C 180,E1 -5553.629,E2 -5553.629} C_VEL
LIN {X 0,Y 509.809,Z 320.603,A -85,B 0,C 180,E1 -5556.436,E2 -5556.436} C_VEL
LIN {X 0,Y 509.903,Z 320.595,A -85,B 0,C 180,E1 -5559.844,E2 -5559.844} C_VEL
LIN {X 0,Y 509.85,Z 320.598,A -85,B 0,C 180,E1 -5563.174,E2 -5563.174} C_VEL
LIN {X 0,Y 509.838,Z 320.605,A -85,B 0,C 180,E1 -5565.634,E2 -5565.634} C_VEL
LIN {X 0,Y 509.875,Z 320.592,A -85,B 0,C 180,E1 -5568.131,E2 -5568.131} C_VEL
LIN {X 0,Y 509.857,Z 320.601,A -85,B 0,C 180,E1 -5571.279,E2 -5571.279} C_VEL
LIN {X 0,Y 509.946,Z 320.584,A -85,B 0,C 180,E1 -5574.464,E2 -5574.464} C_VEL
LIN {X 0,Y 510.028,Z 320.577,A -85,B 0,C 180,E1 -5577.631,E2 -5577.631} C_VEL
LIN {X 0,Y 510.015,Z 320.577,A -85,B 0,C 180,E1 -5580,E2 -5580} C_VEL
LIN {X 0,Y 510.03,Z 320.571,A -85,B 0,C 180,E1 -5582.369,E2 -5582.369} C_VEL
LIN {X 0,Y 509.952,Z 320.588,A -85,B 0,C 180,E1 -5585.536,E2 -5585.536} C_VEL
LIN {X 0,Y 509.907,Z 320.588,A -85,B 0,C 180,E1 -5587.923,E2 -5587.923} C_VEL
LIN {X 0,Y 509.895,Z 320.597,A -85,B 0,C 180,E1 -5591.126,E2 -5591.126} C_VEL
LIN {X 0,Y 509.844,Z 320.598,A -85,B 0,C 180,E1 -5594.367,E2 -5594.367} C_VEL
LIN {X 0,Y 509.866,Z 320.595,A -85,B 0,C 180,E1 -5597.653,E2 -5597.653} C_VEL
LIN {X 0,Y 509.875,Z 320.594,A -85,B 0,C 180,E1 -5600.402,E2 -5600.402} C_VEL
LIN {X 0,Y 509.819,Z 320.6,A -85,B 0,C 180,E1 -5603.564,E2 -5603.564} C_VEL
LIN {X 0,Y 509.901,Z 320.593,A -85,B 0,C 180,E1 -5606.379,E2 -5606.379} C_VEL
LIN {X 0,Y 509.866,Z 320.602,A -85,B 0,C 180,E1 -5608.845,E2 -5608.845} C_VEL
LIN {X 0,Y 509.813,Z 320.599,A -85,B 0,C 180,E1 -5611.591,E2 -5611.591} C_VEL
LIN {X 0,Y 509.843,Z 320.602,A -85,B 0,C 180,E1 -5614.415,E2 -5614.415} C_VEL
LIN {X 0,Y 509.81,Z 320.6,A -85,B 0,C 180,E1 -5617.342,E2 -5617.342} C_VEL
LIN {X 0,Y 509.833,Z 320.604,A -85,B 0,C 180,E1 -5620.383,E2 -5620.383} C_VEL
LIN {X 0,Y 509.819,Z 320.603,A -85,B 0,C 180,E1 -5623.063,E2 -5623.063} C_VEL
LIN {X 0,Y 509.827,Z 320.601,A -85,B 0,C 180,E1 -5625.794,E2 -5625.794} C_VEL
LIN {X 0,Y 509.854,Z 320.603,A -85,B 0,C 180,E1 -5628.576,E2 -5628.576} C_VEL
LIN {X 0,Y 509.85,Z 320.6,A -85,B 0,C 180,E1 -5631.787,E2 -5631.787} C_VEL
LIN {X 0,Y 509.831,Z 320.601,A -85,B 0,C 180,E1 -5633.703,E2 -5633.703} C_VEL
LIN {X 0,Y 509.164,Z 320.688,A -85,B 0,C 180,E1 -5634.363,E2 -5634.363} C_VEL
LIN {X 0,Y 506.35,Z 321.035,A -85,B 0,C 180,E1 -5635.435,E2 -5635.435} C_VEL
LIN {X 0,Y 503.961,Z 321.338,A -85,B 0,C 180,E1 -5636.298,E2 -5636.298} C_VEL
LIN {X 0,Y 502.911,Z 321.465,A -85,B 0,C 180,E1 -5636.964,E2 -5636.964} C_VEL
LIN {X 0,Y 502.812,Z 321.476,A -85,B 0,C 180,E1 -5637.19,E2 -5637.19} C_VEL
LIN {X 0,Y 502.86,Z 321.474,A -85,B 0,C 180,E1 -5640.715,E2 -5640.715} C_VEL
LIN {X 0,Y 504.492,Z 330.088,A -85,B 0,C 180,E1 -5642.407,E2 -5642.407} C_VEL
LIN {X 0,Y 504.188,Z 342.339,A -85,B 0,C 180,E1 -5644.576,E2 -5644.576} C_VEL
LIN {X 0,Y 504.145,Z 344.114,A -85,B 0,C 180,E1 -5644.887,E2 -5644.887} C_VEL
LIN {X 0,Y 506.985,Z 357.525,A -85,B 0,C 180,E1 -5645.213,E2 -5645.213} C_VEL
LIN {X 0,Y 506.129,Z 480.709,A -85,B 0,C 180,E1 -5647.004,E2 -5647.004} C_VEL
LIN {X 0,Y 505.894,Z 495.139,A -85,B 0,C 180,E1 -5647.379,E2 -5647.379} C_VEL
LIN {X 0,Y 505.502,Z 508.88,A -85,B 0,C 180,E1 -5647.899,E2 -5647.899} C_VEL
LIN {X 0,Y 505.081,Z 522.243,A -85,B 0,C 180,E1 -5648.577,E2 -5648.577} C_VEL
LIN {X 0,Y 504.548,Z 535.437,A -85,B 0,C 180,E1 -5649.434,E2 -5649.434} C_VEL
LIN {X 0,Y 504.007,Z 547.922,A -85,B 0,C 180,E1 -5650.449,E2 -5650.449} C_VEL
LIN {X 0,Y 503.65,Z 558.13,A -85,B 0,C 180,E1 -5651.466,E2 -5651.466} C_VEL
LIN {X 0,Y 503.155,Z 568.636,A -85,B 0,C 180,E1 -5652.734,E2 -5652.734} C_VEL
LIN {X 0,Y 502.832,Z 577.119,A -85,B 0,C 180,E1 -5653.976,E2 -5653.976} C_VEL
LIN {X 0,Y 502.542,Z 585.175,A -85,B 0,C 180,E1 -5655.421,E2 -5655.421} C_VEL
LIN {X 0,Y 502.352,Z 590.799,A -85,B 0,C 180,E1 -5656.654,E2 -5656.654} C_VEL
LIN {X 0,Y 502.222,Z 595.377,A -85,B 0,C 180,E1 -5657.883,E2 -5657.883} C_VEL
LIN {X 0,Y 502.163,Z 598.975,A -85,B 0,C 180,E1 -5659.109,E2 -5659.109} C_VEL
LIN {X 0,Y 502.035,Z 601.746,A -85,B 0,C 180,E1 -5660.329,E2 -5660.329} C_VEL
LIN {X 0,Y 502.04,Z 604.153,A -85,B 0,C 180,E1 -5661.953,E2 -5661.953} C_VEL
LIN {X 0,Y 502.15,Z 605.201,A -85,B 0,C 180,E1 -5663.571,E2 -5663.571} C_VEL
LIN {X 0,Y 502.049,Z 604.928,A -85,B 0,C 180,E1 -5665.182,E2 -5665.182} C_VEL
LIN {X 0,Y 502.108,Z 603.33,A -85,B 0,C 180,E1 -5666.791,E2 -5666.791} C_VEL
LIN {X 0,Y 502.052,Z 600.393,A -85,B 0,C 180,E1 -5668.396,E2 -5668.396} C_VEL
LIN {X 0,Y 502.118,Z 596.034,A -85,B 0,C 180,E1 -5670,E2 -5670} C_VEL
LIN {X 0,Y 502.242,Z 590.117,A -85,B 0,C 180,E1 -5671.604,E2 -5671.604} C_VEL
LIN {X 0,Y 502.566,Z 583.463,A -85,B 0,C 180,E1 -5673.006,E2 -5673.006} C_VEL
LIN {X 0,Y 502.851,Z 575.23,A -85,B 0,C 180,E1 -5674.409,E2 -5674.409} C_VEL
LIN {X 0,Y 503.272,Z 566.662,A -85,B 0,C 180,E1 -5675.61,E2 -5675.61} C_VEL
LIN {X 0,Y 503.703,Z 556.318,A -85,B 0,C 180,E1 -5676.811,E2 -5676.811} C_VEL
LIN {X 0,Y 504.172,Z 544.597,A -85,B 0,C 180,E1 -5677.927,E2 -5677.927} C_VEL
LIN {X 0,Y 504.677,Z 533.21,A -85,B 0,C 180,E1 -5678.811,E2 -5678.811} C_VEL
LIN {X 0,Y 505.172,Z 520.507,A -85,B 0,C 180,E1 -5679.61,E2 -5679.61} C_VEL
LIN {X 0,Y 505.589,Z 507.316,A -85,B 0,C 180,E1 -5680.259,E2 -5680.259} C_VEL
LIN {X 0,Y 505.999,Z 493.649,A -85,B 0,C 180,E1 -5680.756,E2 -5680.756} C_VEL
LIN {X 0,Y 506.187,Z 479.445,A -85,B 0,C 180,E1 -5681.107,E2 -5681.107} C_VEL
LIN {X 0,Y 506.918,Z 357.198,A -85,B 0,C 180,E1 -5682.883,E2 -5682.883} C_VEL
LIN {X 0,Y 504.126,Z 344.051,A -85,B 0,C 180,E1 -5683.205,E2 -5683.205} C_VEL
LIN {X 0,Y 504.529,Z 330.693,A -85,B 0,C 180,E1 -5685.548,E2 -5685.548} C_VEL
LIN {X 0,Y 502.857,Z 321.474,A -85,B 0,C 180,E1 -5687.303,E2 -5687.303} C_VEL
LIN {X 0,Y 502.833,Z 321.475,A -85,B 0,C 180,E1 -5690.535,E2 -5690.535} C_VEL
LIN {X 0,Y 502.791,Z 321.477,A -85,B 0,C 180,E1 -5693.04,E2 -5693.04} C_VEL
LIN {X 0,Y 502.824,Z 321.48,A -85,B 0,C 180,E1 -5695.676,E2 -5695.676} C_VEL
LIN {X 0,Y 502.841,Z 321.469,A -85,B 0,C 180,E1 -5698.372,E2 -5698.372} C_VEL
LIN {X 0,Y 502.795,Z 321.482,A -85,B 0,C 180,E1 -5701.498,E2 -5701.498} C_VEL
LIN {X 0,Y 502.805,Z 321.474,A -85,B 0,C 180,E1 -5704.443,E2 -5704.443} C_VEL
LIN {X 0,Y 502.779,Z 321.479,A -85,B 0,C 180,E1 -5707.177,E2 -5707.177} C_VEL
LIN {X 0,Y 502.786,Z 321.472,A -85,B 0,C 180,E1 -5710.014,E2 -5710.014} C_VEL
LIN {X 0,Y 502.8,Z 321.475,A -85,B 0,C 180,E1 -5712.198,E2 -5712.198} C_VEL
LIN {X 0,Y 502.797,Z 321.482,A -85,B 0,C 180,E1 -5715.467,E2 -5715.467} C_VEL
LIN {X 0,Y 502.814,Z 321.474,A -85,B 0,C 180,E1 -5718.933,E2 -5718.933} C_VEL
LIN {X 0,Y 502.786,Z 321.474,A -85,B 0,C 180,E1 -5722.045,E2 -5722.045} C_VEL
LIN {X 0,Y 502.79,Z 321.482,A -85,B 0,C 180,E1 -5725.033,E2 -5725.033} C_VEL
LIN {X 0,Y 502.774,Z 321.478,A -85,B 0,C 180,E1 -5727.914,E2 -5727.914} C_VEL
LIN {X 0,Y 502.813,Z 321.476,A -85,B 0,C 180,E1 -5730.711,E2 -5730.711} C_VEL
LIN {X 0,Y 502.835,Z 321.472,A -85,B 0,C 180,E1 -5733.442,E2 -5733.442} C_VEL
LIN {X 0,Y 502.776,Z 321.485,A -85,B 0,C 180,E1 -5736.958,E2 -5736.958} C_VEL
LIN {X 0,Y 502.822,Z 321.467,A -85,B 0,C 180,E1 -5739.547,E2 -5739.547} C_VEL
LIN {X 0,Y 502.805,Z 321.473,A -85,B 0,C 180,E1 -5742.091,E2 -5742.091} C_VEL
LIN {X 0,Y 502.822,Z 321.47,A -85,B 0,C 180,E1 -5745.428,E2 -5745.428} C_VEL
LIN {X 0,Y 502.86,Z 321.468,A -85,B 0,C 180,E1 -5748.716,E2 -5748.716} C_VEL
LIN {X 0,Y 502.865,Z 321.467,A -85,B 0,C 180,E1 -5751.966,E2 -5751.966} C_VEL
LIN {X 0,Y 502.904,Z 321.463,A -85,B 0,C 180,E1 -5754.386,E2 -5754.386} C_VEL
LIN {X 0,Y 502.997,Z 321.448,A -85,B 0,C 180,E1 -5757.597,E2 -5757.597} C_VEL
LIN {X 0,Y 502.975,Z 321.456,A -85,B 0,C 180,E1 -5760.8,E2 -5760.8} C_VEL
LIN {X 0,Y 502.991,Z 321.455,A -85,B 0,C 180,E1 -5762.402,E2 -5762.402} C_VEL
LIN {X 0,Y 502.888,Z 321.463,A -85,B 0,C 180,E1 -5765.614,E2 -5765.614} C_VEL
LIN {X 0,Y 502.833,Z 321.473,A -85,B 0,C 180,E1 -5768.034,E2 -5768.034} C_VEL
LIN {X 0,Y 502.86,Z 321.466,A -85,B 0,C 180,E1 -5771.283,E2 -5771.283} C_VEL
LIN {X 0,Y 502.828,Z 321.472,A -85,B 0,C 180,E1 -5774.571,E2 -5774.571} C_VEL
LIN {X 0,Y 502.803,Z 321.477,A -85,B 0,C 180,E1 -5777.909,E2 -5777.909} C_VEL
LIN {X 0,Y 502.817,Z 321.471,A -85,B 0,C 180,E1 -5780.536,E2 -5780.536} C_VEL
LIN {X 0,Y 502.775,Z 321.477,A -85,B 0,C 180,E1 -5783.041,E2 -5783.041} C_VEL
LIN {X 0,Y 502.784,Z 321.478,A -85,B 0,C 180,E1 -5785.678,E2 -5785.678} C_VEL
LIN {X 0,Y 502.784,Z 321.479,A -85,B 0,C 180,E1 -5788.376,E2 -5788.376} C_VEL
LIN {X 0,Y 502.785,Z 321.475,A -85,B 0,C 180,E1 -5791.144,E2 -5791.144} C_VEL
LIN {X 0,Y 502.795,Z 321.481,A -85,B 0,C 180,E1 -5793.994,E2 -5793.994} C_VEL
LIN {X 0,Y 502.771,Z 321.479,A -85,B 0,C 180,E1 -5797.179,E2 -5797.179} C_VEL
LIN {X 0,Y 502.779,Z 321.48,A -85,B 0,C 180,E1 -5800.016,E2 -5800.016} C_VEL
LIN {X 0,Y 502.795,Z 321.477,A -85,B 0,C 180,E1 -5802.2,E2 -5802.2} C_VEL
LIN {X 0,Y 502.794,Z 321.481,A -85,B 0,C 180,E1 -5805.469,E2 -5805.469} C_VEL
LIN {X 0,Y 502.814,Z 321.474,A -85,B 0,C 180,E1 -5808.935,E2 -5808.935} C_VEL
LIN {X 0,Y 502.789,Z 321.481,A -85,B 0,C 180,E1 -5812.047,E2 -5812.047} C_VEL
LIN {X 0,Y 502.803,Z 321.48,A -85,B 0,C 180,E1 -5815.036,E2 -5815.036} C_VEL
LIN {X 0,Y 502.781,Z 321.482,A -85,B 0,C 180,E1 -5817.916,E2 -5817.916} C_VEL
LIN {X 0,Y 502.821,Z 321.475,A -85,B 0,C 180,E1 -5820.713,E2 -5820.713} C_VEL
LIN {X 0,Y 502.861,Z 321.531,A -85,B 0,C 180,E1 -5823.389,E2 -5823.389} C_VEL
LIN {X 0,Y 505.325,Z 333.398,A -85,B 0,C 180,E1 -5825.341,E2 -5825.341} C_VEL
LIN {X 0,Y 504.896,Z 347.69,A -85,B 0,C 180,E1 -5827.494,E2 -5827.494} C_VEL
LIN {X 0,Y 504.211,Z 369.289,A -85,B 0,C 180,E1 -5830.706,E2 -5830.706} C_VEL
LIN {X 0,Y 504.161,Z 370.173,A -85,B 0,C 180,E1 -5830.836,E2 -5830.836} C_VEL
LIN {X 0,Y 506.961,Z 387.095,A -85,B 0,C 180,E1 -5831.202,E2 -5831.202} C_VEL
LIN {X 0,Y 506.038,Z 508.603,A -85,B 0,C 180,E1 -5832.966,E2 -5832.966} C_VEL
LIN {X 0,Y 505.698,Z 523.13,A -85,B 0,C 180,E1 -5833.343,E2 -5833.343} C_VEL
LIN {X 0,Y 505.368,Z 536.499,A -85,B 0,C 180,E1 -5833.852,E2 -5833.852} C_VEL
LIN {X 0,Y 504.898,Z 550.474,A -85,B 0,C 180,E1 -5834.561,E2 -5834.561} C_VEL
LIN {X 0,Y 504.357,Z 562.978,A -85,B 0,C 180,E1 -5835.371,E2 -5835.371} C_VEL
LIN {X 0,Y 503.835,Z 575.584,A -85,B 0,C 180,E1 -5836.386,E2 -5836.386} C_VEL
LIN {X 0,Y 503.434,Z 586.18,A -85,B 0,C 180,E1 -5837.432,E2 -5837.432} C_VEL
LIN {X 0,Y 503.028,Z 596.895,A -85,B 0,C 180,E1 -5838.721,E2 -5838.721} C_VEL
LIN {X 0,Y 502.702,Z 605.265,A -85,B 0,C 180,E1 -5839.936,E2 -5839.936} C_VEL
LIN {X 0,Y 502.437,Z 613.268,A -85,B 0,C 180,E1 -5841.352,E2 -5841.352} C_VEL
LIN {X 0,Y 502.252,Z 619.714,A -85,B 0,C 180,E1 -5842.765,E2 -5842.765} C_VEL
LIN {X 0,Y 502.2,Z 625.43,A -85,B 0,C 180,E1 -5844.378,E2 -5844.378} C_VEL
LIN {X 0,Y 502.112,Z 629.575,A -85,B 0,C 180,E1 -5845.987,E2 -5845.987} C_VEL
LIN {X 0,Y 502.089,Z 632.283,A -85,B 0,C 180,E1 -5847.593,E2 -5847.593} C_VEL
LIN {X 0,Y 501.988,Z 633.622,A -85,B 0,C 180,E1 -5849.198,E2 -5849.198} C_VEL
LIN {X 0,Y 501.988,Z 633.622,A -85,B 0,C 180,E1 -5850.802,E2 -5850.802} C_VEL
LIN {X 0,Y 502.089,Z 632.282,A -85,B 0,C 180,E1 -5852.407,E2 -5852.407} C_VEL
LIN {X 0,Y 502.112,Z 629.573,A -85,B 0,C 180,E1 -5854.013,E2 -5854.013} C_VEL
LIN {X 0,Y 502.2,Z 625.421,A -85,B 0,C 180,E1 -5855.622,E2 -5855.622} C_VEL
LIN {X 0,Y 502.252,Z 619.699,A -85,B 0,C 180,E1 -5857.235,E2 -5857.235} C_VEL
LIN {X 0,Y 502.438,Z 613.253,A -85,B 0,C 180,E1 -5858.648,E2 -5858.648} C_VEL
LIN {X 0,Y 502.685,Z 605.245,A -85,B 0,C 180,E1 -5860.065,E2 -5860.065} C_VEL
LIN {X 0,Y 503.024,Z 596.873,A -85,B 0,C 180,E1 -5861.28,E2 -5861.28} C_VEL
LIN {X 0,Y 503.414,Z 586.154,A -85,B 0,C 180,E1 -5862.568,E2 -5862.568} C_VEL
LIN {X 0,Y 503.853,Z 575.555,A -85,B 0,C 180,E1 -5863.614,E2 -5863.614} C_VEL
LIN {X 0,Y 504.326,Z 564.379,A -85,B 0,C 180,E1 -5864.527,E2 -5864.527} C_VEL
LIN {X 0,Y 504.799,Z 552.211,A -85,B 0,C 180,E1 -5865.338,E2 -5865.338} C_VEL
LIN {X 0,Y 505.319,Z 538.716,A -85,B 0,C 180,E1 -5866.046,E2 -5866.046} C_VEL
LIN {X 0,Y 505.662,Z 524.604,A -85,B 0,C 180,E1 -5866.606,E2 -5866.606} C_VEL
LIN {X 0,Y 506.01,Z 510.839,A -85,B 0,C 180,E1 -5866.983,E2 -5866.983} C_VEL
LIN {X 0,Y 506.18,Z 490.515,A -85,B 0,C 180,E1 -5867.316,E2 -5867.316} C_VEL
LIN {X 0,Y 506.903,Z 386.441,A -85,B 0,C 180,E1 -5868.81,E2 -5868.81} C_VEL
LIN {X 0,Y 504.186,Z 370.139,A -85,B 0,C 180,E1 -5869.163,E2 -5869.163} C_VEL
LIN {X 0,Y 504.874,Z 347.735,A -85,B 0,C 180,E1 -5872.507,E2 -5872.507} C_VEL
LIN {X 0,Y 505.391,Z 333.593,A -85,B 0,C 180,E1 -5874.656,E2 -5874.656} C_VEL
LIN {X 0,Y 502.85,Z 321.476,A -85,B 0,C 180,E1 -5876.717,E2 -5876.717} C_VEL
LIN {X 0,Y 502.821,Z 321.476,A -85,B 0,C 180,E1 -5879.287,E2 -5879.287} C_VEL
LIN {X 0,Y 502.78,Z 321.483,A -85,B 0,C 180,E1 -5882.084,E2 -5882.084} C_VEL
LIN {X 0,Y 502.803,Z 321.477,A -85,B 0,C 180,E1 -5884.964,E2 -5884.964} C_VEL
LIN {X 0,Y 502.789,Z 321.474,A -85,B 0,C 180,E1 -5887.953,E2 -5887.953} C_VEL
LIN {X 0,Y 502.814,Z 321.471,A -85,B 0,C 180,E1 -5891.065,E2 -5891.065} C_VEL
LIN {X 0,Y 502.794,Z 321.478,A -85,B 0,C 180,E1 -5894.531,E2 -5894.531} C_VEL
LIN {X 0,Y 502.788,Z 321.478,A -85,B 0,C 180,E1 -5897.86,E2 -5897.86} C_VEL
LIN {X 0,Y 502.792,Z 321.476,A -85,B 0,C 180,E1 -5901.023,E2 -5901.023} C_VEL
LIN {X 0,Y 502.772,Z 321.485,A -85,B 0,C 180,E1 -5904.167,E2 -5904.167} C_VEL
LIN {X 0,Y 502.822,Z 321.472,A -85,B 0,C 180,E1 -5906.993,E2 -5906.993} C_VEL
LIN {X 0,Y 502.804,Z 321.47,A -85,B 0,C 180,E1 -5910.064,E2 -5910.064} C_VEL
LIN {X 0,Y 502.832,Z 321.473,A -85,B 0,C 180,E1 -5913.443,E2 -5913.443} C_VEL
LIN {X 0,Y 502.761,Z 321.485,A -85,B 0,C 180,E1 -5916.085,E2 -5916.085} C_VEL
LIN {X 0,Y 502.77,Z 321.477,A -85,B 0,C 180,E1 -5918.688,E2 -5918.688} C_VEL
LIN {X 0,Y 502.809,Z 321.475,A -85,B 0,C 180,E1 -5921.248,E2 -5921.248} C_VEL
LIN {X 0,Y 502.835,Z 321.469,A -85,B 0,C 180,E1 -5924.6,E2 -5924.6} C_VEL
LIN {X 0,Y 502.855,Z 321.467,A -85,B 0,C 180,E1 -5928.043,E2 -5928.043} C_VEL
LIN {X 0,Y 502.82,Z 321.476,A -85,B 0,C 180,E1 -5931.156,E2 -5931.156} C_VEL
LIN {X 0,Y 502.854,Z 321.473,A -85,B 0,C 180,E1 -5933.581,E2 -5933.581} C_VEL
LIN {X 0,Y 502.839,Z 321.47,A -85,B 0,C 180,E1 -5936.795,E2 -5936.795} C_VEL
LIN {X 0,Y 502.876,Z 321.462,A -85,B 0,C 180,E1 -5938.399,E2 -5938.399} C_VEL
LIN {X 0,Y 502.984,Z 321.453,A -85,B 0,C 180,E1 -5940,E2 -5940} C_VEL
LIN {X 0,Y 502.999,Z 321.447,A -85,B 0,C 180,E1 -5942.403,E2 -5942.403} C_VEL
LIN {X 0,Y 502.906,Z 321.464,A -85,B 0,C 180,E1 -5945.614,E2 -5945.614} C_VEL
LIN {X 0,Y 502.866,Z 321.465,A -85,B 0,C 180,E1 -5948.034,E2 -5948.034} C_VEL
LIN {X 0,Y 502.861,Z 321.47,A -85,B 0,C 180,E1 -5951.284,E2 -5951.284} C_VEL
LIN {X 0,Y 502.823,Z 321.474,A -85,B 0,C 180,E1 -5954.572,E2 -5954.572} C_VEL
LIN {X 0,Y 502.807,Z 321.479,A -85,B 0,C 180,E1 -5957.07,E2 -5957.07} C_VEL
LIN {X 0,Y 502.812,Z 321.473,A -85,B 0,C 180,E1 -5959.601,E2 -5959.601} C_VEL
LIN {X 0,Y 502.793,Z 321.481,A -85,B 0,C 180,E1 -5962.703,E2 -5962.703} C_VEL
LIN {X 0,Y 502.83,Z 321.471,A -85,B 0,C 180,E1 -5965.677,E2 -5965.677} C_VEL
LIN {X 0,Y 502.83,Z 321.472,A -85,B 0,C 180,E1 -5968.374,E2 -5968.374} C_VEL
LIN {X 0,Y 502.786,Z 321.475,A -85,B 0,C 180,E1 -5971.5,E2 -5971.5} C_VEL
LIN {X 0,Y 502.798,Z 321.475,A -85,B 0,C 180,E1 -5973.995,E2 -5973.995} C_VEL
LIN {X 0,Y 502.771,Z 321.478,A -85,B 0,C 180,E1 -5977.179,E2 -5977.179} C_VEL
LIN {X 0,Y 502.783,Z 321.478,A -85,B 0,C 180,E1 -5980.016,E2 -5980.016} C_VEL
LIN {X 0,Y 502.798,Z 321.48,A -85,B 0,C 180,E1 -5982.2,E2 -5982.2} C_VEL
LIN {X 0,Y 502.797,Z 321.476,A -85,B 0,C 180,E1 -5985.469,E2 -5985.469} C_VEL
LIN {X 0,Y 502.818,Z 321.476,A -85,B 0,C 180,E1 -5988.935,E2 -5988.935} C_VEL
LIN {X 0,Y 502.793,Z 321.482,A -85,B 0,C 180,E1 -5992.047,E2 -5992.047} C_VEL
LIN {X 0,Y 502.808,Z 321.473,A -85,B 0,C 180,E1 -5995.036,E2 -5995.036} C_VEL
LIN {X 0,Y 502.812,Z 321.476,A -85,B 0,C 180,E1 -5997.19,E2 -5997.19} C_VEL
LIN {X 0,Y 502.11,Z 321.566,A -85,B 0,C 180,E1 -5997.636,E2 -5997.636} C_VEL
LIN {X 0,Y 496.418,Z 322.275,A -85,B 0,C 180,E1 -5999.038,E2 -5999.038} C_VEL
LIN {X 0,Y 495.752,Z 322.357,A -85,B 0,C 180,E1 -5999.493,E2 -5999.493} C_VEL
LIN {X 0,Y 495.827,Z 322.518,A -85,B 0,C 180,E1 -6000.55,E2 -6000.55} C_VEL
LIN {X 0,Y 497.631,Z 332.06,A -85,B 0,C 180,E1 -6002.407,E2 -6002.407} C_VEL
LIN {X 0,Y 497.255,Z 344.535,A -85,B 0,C 180,E1 -6004.622,E2 -6004.622} C_VEL
LIN {X 0,Y 500.337,Z 359.397,A -85,B 0,C 180,E1 -6004.974,E2 -6004.974} C_VEL
LIN {X 0,Y 499.347,Z 481.195,A -85,B 0,C 180,E1 -6006.771,E2 -6006.771} C_VEL
LIN {X 0,Y 499.092,Z 495.868,A -85,B 0,C 180,E1 -6007.163,E2 -6007.163} C_VEL
LIN {X 0,Y 498.678,Z 509.466,A -85,B 0,C 180,E1 -6007.689,E2 -6007.689} C_VEL
LIN {X 0,Y 498.223,Z 522.737,A -85,B 0,C 180,E1 -6008.376,E2 -6008.376} C_VEL
LIN {X 0,Y 497.703,Z 534.771,A -85,B 0,C 180,E1 -6009.165,E2 -6009.165} C_VEL
LIN {X 0,Y 497.162,Z 547.124,A -85,B 0,C 180,E1 -6010.168,E2 -6010.168} C_VEL
LIN {X 0,Y 496.697,Z 558.655,A -85,B 0,C 180,E1 -6011.323,E2 -6011.323} C_VEL
LIN {X 0,Y 496.217,Z 568.203,A -85,B 0,C 180,E1 -6012.485,E2 -6012.485} C_VEL
LIN {X 0,Y 495.845,Z 576.796,A -85,B 0,C 180,E1 -6013.744,E2 -6013.744} C_VEL
LIN {X 0,Y 495.495,Z 584.948,A -85,B 0,C 180,E1 -6015.209,E2 -6015.209} C_VEL
LIN {X 0,Y 495.316,Z 590.66,A -85,B 0,C 180,E1 -6016.461,E2 -6016.461} C_VEL
LIN {X 0,Y 495.157,Z 595.278,A -85,B 0,C 180,E1 -6017.708,E2 -6017.708} C_VEL
LIN {X 0,Y 495.098,Z 598.953,A -85,B 0,C 180,E1 -6018.952,E2 -6018.952} C_VEL
LIN {X 0,Y 494.969,Z 601.795,A -85,B 0,C 180,E1 -6020.19,E2 -6020.19} C_VEL
LIN {X 0,Y 494.956,Z 604.271,A -85,B 0,C 180,E1 -6021.837,E2 -6021.837} C_VEL
LIN {X 0,Y 495.063,Z 605.406,A -85,B 0,C 180,E1 -6023.586,E2 -6023.586} C_VEL
LIN {X 0,Y 494.971,Z 605.179,A -85,B 0,C 180,E1 -6025.113,E2 -6025.113} C_VEL
LIN {X 0,Y 495.028,Z 603.647,A -85,B 0,C 180,E1 -6026.745,E2 -6026.745} C_VEL
LIN {X 0,Y 494.978,Z 600.778,A -85,B 0,C 180,E1 -6028.373,E2 -6028.373} C_VEL
LIN {X 0,Y 495.033,Z 596.492,A -85,B 0,C 180,E1 -6030,E2 -6030} C_VEL
LIN {X 0,Y 495.167,Z 590.667,A -85,B 0,C 180,E1 -6031.627,E2 -6031.627} C_VEL
LIN {X 0,Y 495.513,Z 584.108,A -85,B 0,C 180,E1 -6033.049,E2 -6033.049} C_VEL
LIN {X 0,Y 495.818,Z 575.989,A -85,B 0,C 180,E1 -6034.471,E2 -6034.471} C_VEL
LIN {X 0,Y 496.272,Z 567.531,A -85,B 0,C 180,E1 -6035.689,E2 -6035.689} C_VEL
LIN {X 0,Y 496.729,Z 557.319,A -85,B 0,C 180,E1 -6036.907,E2 -6036.907} C_VEL
LIN {X 0,Y 497.153,Z 547.248,A -85,B 0,C 180,E1 -6037.908,E2 -6037.908} C_VEL
LIN {X 0,Y 497.668,Z 535.987,A -85,B 0,C 180,E1 -6038.834,E2 -6038.834} C_VEL
LIN {X 0,Y 498.207,Z 523.887,A -85,B 0,C 180,E1 -6039.643,E2 -6039.643} C_VEL
LIN {X 0,Y 498.687,Z 510.47,A -85,B 0,C 180,E1 -6040.351,E2 -6040.351} C_VEL
LIN {X 0,Y 499.091,Z 496.377,A -85,B 0,C 180,E1 -6040.907,E2 -6040.907} C_VEL
LIN {X 0,Y 499.391,Z 482.442,A -85,B 0,C 180,E1 -6041.286,E2 -6041.286} C_VEL
LIN {X 0,Y 499.613,Z 453.232,A -85,B 0,C 180,E1 -6041.743,E2 -6041.743} C_VEL
LIN {X 0,Y 500.21,Z 358.256,A -85,B 0,C 180,E1 -6043.13,E2 -6043.13} C_VEL
LIN {X 0,Y 497.235,Z 344.27,A -85,B 0,C 180,E1 -6043.47,E2 -6043.47} C_VEL
LIN {X 0,Y 497.615,Z 332.45,A -85,B 0,C 180,E1 -6045.565,E2 -6045.565} C_VEL
LIN {X 0,Y 496.214,Z 324.411,A -85,B 0,C 180,E1 -6047.09,E2 -6047.09} C_VEL
LIN {X 0,Y 495.818,Z 322.352,A -85,B 0,C 180,E1 -6047.53,E2 -6047.53} C_VEL
LIN {X 0,Y 495.778,Z 322.353,A -85,B 0,C 180,E1 -6050.756,E2 -6050.756} C_VEL
LIN {X 0,Y 495.746,Z 322.357,A -85,B 0,C 180,E1 -6053.387,E2 -6053.387} C_VEL
LIN {X 0,Y 495.826,Z 322.345,A -85,B 0,C 180,E1 -6056.748,E2 -6056.748} C_VEL
LIN {X 0,Y 495.768,Z 322.358,A -85,B 0,C 180,E1 -6059.745,E2 -6059.745} C_VEL
LIN {X 0,Y 495.769,Z 322.35,A -85,B 0,C 180,E1 -6062.593,E2 -6062.593} C_VEL
LIN {X 0,Y 495.756,Z 322.356,A -85,B 0,C 180,E1 -6065.536,E2 -6065.536} C_VEL
LIN {X 0,Y 495.762,Z 322.352,A -85,B 0,C 180,E1 -6068.767,E2 -6068.767} C_VEL
LIN {X 0,Y 495.753,Z 322.357,A -85,B 0,C 180,E1 -6071.78,E2 -6071.78} C_VEL
LIN {X 0,Y 495.746,Z 322.357,A -85,B 0,C 180,E1 -6075.138,E2 -6075.138} C_VEL
LIN {X 0,Y 495.751,Z 322.35,A -85,B 0,C 180,E1 -6078.218,E2 -6078.218} C_VEL
LIN {X 0,Y 495.744,Z 322.358,A -85,B 0,C 180,E1 -6081.407,E2 -6081.407} C_VEL
LIN {X 0,Y 495.741,Z 322.354,A -85,B 0,C 180,E1 -6084.461,E2 -6084.461} C_VEL
LIN {X 0,Y 495.758,Z 322.357,A -85,B 0,C 180,E1 -6087.404,E2 -6087.404} C_VEL
LIN {X 0,Y 495.757,Z 322.352,A -85,B 0,C 180,E1 -6090.253,E2 -6090.253} C_VEL
LIN {X 0,Y 495.796,Z 322.35,A -85,B 0,C 180,E1 -6093.254,E2 -6093.254} C_VEL
LIN {X 0,Y 495.729,Z 322.359,A -85,B 0,C 180,E1 -6096.611,E2 -6096.611} C_VEL
LIN {X 0,Y 495.768,Z 322.347,A -85,B 0,C 180,E1 -6099.323,E2 -6099.323} C_VEL
LIN {X 0,Y 495.767,Z 322.349,A -85,B 0,C 180,E1 -6101.828,E2 -6101.828} C_VEL
LIN {X 0,Y 495.812,Z 322.349,A -85,B 0,C 180,E1 -6104.548,E2 -6104.548} C_VEL
LIN {X 0,Y 495.816,Z 322.337,A -85,B 0,C 180,E1 -6107.965,E2 -6107.965} C_VEL
LIN {X 0,Y 495.816,Z 322.349,A -85,B 0,C 180,E1 -6111.029,E2 -6111.029} C_VEL
LIN {X 0,Y 495.834,Z 322.34,A -85,B 0,C 180,E1 -6113.489,E2 -6113.489} C_VEL
LIN {X 0,Y 495.797,Z 322.349,A -85,B 0,C 180,E1 -6116.749,E2 -6116.749} C_VEL
LIN {X 0,Y 495.856,Z 322.343,A -85,B 0,C 180,E1 -6118.375,E2 -6118.375} C_VEL
LIN {X 0,Y 495.927,Z 322.334,A -85,B 0,C 180,E1 -6120.812,E2 -6120.812} C_VEL
LIN {X 0,Y 495.958,Z 322.33,A -85,B 0,C 180,E1 -6122.436,E2 -6122.436} C_VEL
LIN {X 0,Y 495.845,Z 322.341,A -85,B 0,C 180,E1 -6125.694,E2 -6125.694} C_VEL
LIN {X 0,Y 495.798,Z 322.351,A -85,B 0,C 180,E1 -6128.149,E2 -6128.149} C_VEL
LIN {X 0,Y 495.836,Z 322.341,A -85,B 0,C 180,E1 -6131.445,E2 -6131.445} C_VEL
LIN {X 0,Y 495.774,Z 322.348,A -85,B 0,C 180,E1 -6134.783,E2 -6134.783} C_VEL
LIN {X 0,Y 495.744,Z 322.352,A -85,B 0,C 180,E1 -6137.32,E2 -6137.32} C_VEL
LIN {X 0,Y 495.754,Z 322.356,A -85,B 0,C 180,E1 -6139.891,E2 -6139.891} C_VEL
LIN {X 0,Y 495.746,Z 322.353,A -85,B 0,C 180,E1 -6142.861,E2 -6142.861} C_VEL
LIN {X 0,Y 495.747,Z 322.357,A -85,B 0,C 180,E1 -6146.07,E2 -6146.07} C_VEL
LIN {X 0,Y 495.732,Z 322.355,A -85,B 0,C 180,E1 -6148.817,E2 -6148.817} C_VEL
LIN {X 0,Y 495.744,Z 322.357,A -85,B 0,C 180,E1 -6151.726,E2 -6151.726} C_VEL
LIN {X 0,Y 495.762,Z 322.351,A -85,B 0,C 180,E1 -6154.695,E2 -6154.695} C_VEL
LIN {X 0,Y 495.721,Z 322.361,A -85,B 0,C 180,E1 -6157.562,E2 -6157.562} C_VEL
LIN {X 0,Y 495.758,Z 322.349,A -85,B 0,C 180,E1 -6160.701,E2 -6160.701} C_VEL
LIN {X 0,Y 495.726,Z 322.36,A -85,B 0,C 180,E1 -6164.002,E2 -6164.002} C_VEL
LIN {X 0,Y 495.719,Z 322.359,A -85,B 0,C 180,E1 -6167.118,E2 -6167.118} C_VEL
LIN {X 0,Y 495.753,Z 322.358,A -85,B 0,C 180,E1 -6169.954,E2 -6169.954} C_VEL
LIN {X 0,Y 495.725,Z 322.359,A -85,B 0,C 180,E1 -6172.554,E2 -6172.554} C_VEL
LIN {X 0,Y 495.779,Z 322.358,A -85,B 0,C 180,E1 -6175.458,E2 -6175.458} C_VEL
LIN {X 0,Y 495.753,Z 322.355,A -85,B 0,C 180,E1 -6178.365,E2 -6178.365} C_VEL
LIN {X 0,Y 495.785,Z 322.354,A -85,B 0,C 180,E1 -6181.508,E2 -6181.508} C_VEL
LIN {X 0,Y 495.826,Z 322.5,A -85,B 0,C 180,E1 -6183.182,E2 -6183.182} C_VEL
LIN {X 0,Y 498.377,Z 334.553,A -85,B 0,C 180,E1 -6185.196,E2 -6185.196} C_VEL
LIN {X 0,Y 498.186,Z 342.963,A -85,B 0,C 180,E1 -6186.487,E2 -6186.487} C_VEL
LIN {X 0,Y 497.568,Z 359.845,A -85,B 0,C 180,E1 -6189.041,E2 -6189.041} C_VEL
LIN {X 0,Y 497.253,Z 370.017,A -85,B 0,C 180,E1 -6190.569,E2 -6190.569} C_VEL
LIN {X 0,Y 500.229,Z 387.861,A -85,B 0,C 180,E1 -6190.954,E2 -6190.954} C_VEL
LIN {X 0,Y 499.261,Z 508.389,A -85,B 0,C 180,E1 -6192.727,E2 -6192.727} C_VEL
LIN {X 0,Y 498.917,Z 522.644,A -85,B 0,C 180,E1 -6193.101,E2 -6193.101} C_VEL
LIN {X 0,Y 498.534,Z 536.292,A -85,B 0,C 180,E1 -6193.624,E2 -6193.624} C_VEL
LIN {X 0,Y 498.029,Z 550.268,A -85,B 0,C 180,E1 -6194.343,E2 -6194.343} C_VEL
LIN {X 0,Y 497.431,Z 562.772,A -85,B 0,C 180,E1 -6195.163,E2 -6195.163} C_VEL
LIN {X 0,Y 496.927,Z 575.38,A -85,B 0,C 180,E1 -6196.193,E2 -6196.193} C_VEL
LIN {X 0,Y 496.429,Z 585.975,A -85,B 0,C 180,E1 -6197.252,E2 -6197.252} C_VEL
LIN {X 0,Y 496.054,Z 595.315,A -85,B 0,C 180,E1 -6198.372,E2 -6198.372} C_VEL
LIN {X 0,Y 495.709,Z 603.789,A -85,B 0,C 180,E1 -6199.586,E2 -6199.586} C_VEL
LIN {X 0,Y 495.402,Z 612.051,A -85,B 0,C 180,E1 -6201.023,E2 -6201.023} C_VEL
LIN {X 0,Y 495.209,Z 617.834,A -85,B 0,C 180,E1 -6202.252,E2 -6202.252} C_VEL
LIN {X 0,Y 495.118,Z 623.57,A -85,B 0,C 180,E1 -6203.764,E2 -6203.764} C_VEL
LIN {X 0,Y 495.03,Z 627.487,A -85,B 0,C 180,E1 -6205.114,E2 -6205.114} C_VEL
LIN {X 0,Y 495.033,Z 630.903,A -85,B 0,C 180,E1 -6206.745,E2 -6206.745} C_VEL
LIN {X 0,Y 494.959,Z 632.921,A -85,B 0,C 180,E1 -6208.373,E2 -6208.373} C_VEL
LIN {X 0,Y 494.896,Z 633.588,A -85,B 0,C 180,E1 -6210,E2 -6210} C_VEL
LIN {X 0,Y 494.959,Z 632.919,A -85,B 0,C 180,E1 -6211.627,E2 -6211.627} C_VEL
LIN {X 0,Y 495.033,Z 630.9,A -85,B 0,C 180,E1 -6213.255,E2 -6213.255} C_VEL
LIN {X 0,Y 495.03,Z 627.48,A -85,B 0,C 180,E1 -6214.886,E2 -6214.886} C_VEL
LIN {X 0,Y 495.129,Z 622.678,A -85,B 0,C 180,E1 -6216.486,E2 -6216.486} C_VEL
LIN {X 0,Y 495.209,Z 617.816,A -85,B 0,C 180,E1 -6217.748,E2 -6217.748} C_VEL
LIN {X 0,Y 495.44,Z 610.939,A -85,B 0,C 180,E1 -6219.183,E2 -6219.183} C_VEL
LIN {X 0,Y 495.772,Z 602.403,A -85,B 0,C 180,E1 -6220.619,E2 -6220.619} C_VEL
LIN {X 0,Y 496.146,Z 592.805,A -85,B 0,C 180,E1 -6221.94,E2 -6221.94} C_VEL
LIN {X 0,Y 496.544,Z 582.716,A -85,B 0,C 180,E1 -6223.088,E2 -6223.088} C_VEL
LIN {X 0,Y 497.017,Z 571.81,A -85,B 0,C 180,E1 -6224.118,E2 -6224.118} C_VEL
LIN {X 0,Y 497.602,Z 559.878,A -85,B 0,C 180,E1 -6225.041,E2 -6225.041} C_VEL
LIN {X 0,Y 498.148,Z 546.673,A -85,B 0,C 180,E1 -6225.863,E2 -6225.863} C_VEL
LIN {X 0,Y 498.625,Z 532.758,A -85,B 0,C 180,E1 -6226.527,E2 -6226.527} C_VEL
LIN {X 0,Y 498.974,Z 518.617,A -85,B 0,C 180,E1 -6227.021,E2 -6227.021} C_VEL
LIN {X 0,Y 499.309,Z 504.077,A -85,B 0,C 180,E1 -6227.35,E2 -6227.35} C_VEL
LIN {X 0,Y 500.189,Z 387.721,A -85,B 0,C 180,E1 -6229.052,E2 -6229.052} C_VEL
LIN {X 0,Y 497.229,Z 369.964,A -85,B 0,C 180,E1 -6229.442,E2 -6229.442} C_VEL
LIN {X 0,Y 497.912,Z 350.453,A -85,B 0,C 180,E1 -6232.401,E2 -6232.401} C_VEL
LIN {X 0,Y 498.492,Z 334.929,A -85,B 0,C 180,E1 -6234.798,E2 -6234.798} C_VEL
LIN {X 0,Y 495.819,Z 322.351,A -85,B 0,C 180,E1 -6236.973,E2 -6236.973} C_VEL
LIN {X 0,Y 495.762,Z 322.357,A -85,B 0,C 180,E1 -6240.146,E2 -6240.146} C_VEL
LIN {X 0,Y 495.789,Z 322.351,A -85,B 0,C 180,E1 -6243.244,E2 -6243.244} C_VEL
LIN {X 0,Y 495.723,Z 322.36,A -85,B 0,C 180,E1 -6246.089,E2 -6246.089} C_VEL
LIN {X 0,Y 495.758,Z 322.354,A -85,B 0,C 180,E1 -6248.767,E2 -6248.767} C_VEL
LIN {X 0,Y 495.751,Z 322.351,A -85,B 0,C 180,E1 -6251.78,E2 -6251.78} C_VEL
LIN {X 0,Y 495.742,Z 322.351,A -85,B 0,C 180,E1 -6255.139,E2 -6255.139} C_VEL
LIN {X 0,Y 495.749,Z 322.359,A -85,B 0,C 180,E1 -6258.218,E2 -6258.218} C_VEL
LIN {X 0,Y 495.741,Z 322.355,A -85,B 0,C 180,E1 -6261.408,E2 -6261.408} C_VEL
LIN {X 0,Y 495.744,Z 322.356,A -85,B 0,C 180,E1 -6264.462,E2 -6264.462} C_VEL
LIN {X 0,Y 495.757,Z 322.353,A -85,B 0,C 180,E1 -6267.405,E2 -6267.405} C_VEL
LIN {X 0,Y 495.752,Z 322.348,A -85,B 0,C 180,E1 -6270.253,E2 -6270.253} C_VEL
LIN {X 0,Y 495.762,Z 322.352,A -85,B 0,C 180,E1 -6273.262,E2 -6273.262} C_VEL
LIN {X 0,Y 495.729,Z 322.356,A -85,B 0,C 180,E1 -6276.612,E2 -6276.612} C_VEL
LIN {X 0,Y 495.766,Z 322.352,A -85,B 0,C 180,E1 -6279.324,E2 -6279.324} C_VEL
LIN {X 0,Y 495.766,Z 322.358,A -85,B 0,C 180,E1 -6281.828,E2 -6281.828} C_VEL
LIN {X 0,Y 495.81,Z 322.344,A -85,B 0,C 180,E1 -6284.549,E2 -6284.549} C_VEL
LIN {X 0,Y 495.808,Z 322.346,A -85,B 0,C 180,E1 -6287.969,E2 -6287.969} C_VEL
LIN {X 0,Y 495.762,Z 322.354,A -85,B 0,C 180,E1 -6291.029,E2 -6291.029} C_VEL
LIN {X 0,Y 495.805,Z 322.35,A -85,B 0,C 180,E1 -6293.489,E2 -6293.489} C_VEL
LIN {X 0,Y 495.687,Z 322.363,A -85,B 0,C 180,E1 -6295.935,E2 -6295.935} C_VEL
LIN {X 0,Y 495.965,Z 322.329,A -85,B 0,C 180,E1 -6297.564,E2 -6297.564} C_VEL
LIN {X 0,Y 495.954,Z 322.329,A -85,B 0,C 180,E1 -6300,E2 -6300} C_VEL
LIN {X 0,Y 495.968,Z 322.323,A -85,B 0,C 180,E1 -6302.437,E2 -6302.437} C_VEL
LIN {X 0,Y 495.863,Z 322.341,A -85,B 0,C 180,E1 -6305.694,E2 -6305.694} C_VEL
LIN {X 0,Y 495.822,Z 322.342,A -85,B 0,C 180,E1 -6308.149,E2 -6308.149} C_VEL
LIN {X 0,Y 495.836,Z 322.342,A -85,B 0,C 180,E1 -6311.446,E2 -6311.446} C_VEL
LIN {X 0,Y 495.771,Z 322.355,A -85,B 0,C 180,E1 -6314.784,E2 -6314.784} C_VEL
LIN {X 0,Y 495.752,Z 322.357,A -85,B 0,C 180,E1 -6317.32,E2 -6317.32} C_VEL
LIN {X 0,Y 495.759,Z 322.351,A -85,B 0,C 180,E1 -6319.891,E2 -6319.891} C_VEL
LIN {X 0,Y 495.749,Z 322.361,A -85,B 0,C 180,E1 -6322.861,E2 -6322.861} C_VEL
LIN {X 0,Y 495.781,Z 322.35,A -85,B 0,C 180,E1 -6326.069,E2 -6326.069} C_VEL
LIN {X 0,Y 495.763,Z 322.357,A -85,B 0,C 180,E1 -6328.816,E2 -6328.816} C_VEL
LIN {X 0,Y 495.748,Z 322.351,A -85,B 0,C 180,E1 -6331.726,E2 -6331.726} C_VEL
LIN {X 0,Y 495.764,Z 322.356,A -85,B 0,C 180,E1 -6334.695,E2 -6334.695} C_VEL
LIN {X 0,Y 495.723,Z 322.355,A -85,B 0,C 180,E1 -6337.563,E2 -6337.563} C_VEL
LIN {X 0,Y 495.762,Z 322.358,A -85,B 0,C 180,E1 -6340.701,E2 -6340.701} C_VEL
LIN {X 0,Y 495.731,Z 322.359,A -85,B 0,C 180,E1 -6344.002,E2 -6344.002} C_VEL
LIN {X 0,Y 495.722,Z 322.358,A -85,B 0,C 180,E1 -6347.118,E2 -6347.118} C_VEL
LIN {X 0,Y 495.757,Z 322.357,A -85,B 0,C 180,E1 -6349.954,E2 -6349.954} C_VEL
LIN {X 0,Y 495.729,Z 322.361,A -85,B 0,C 180,E1 -6352.554,E2 -6352.554} C_VEL
LIN {X 0,Y 495.784,Z 322.348,A -85,B 0,C 180,E1 -6355.458,E2 -6355.458} C_VEL
LIN {X 0,Y 495.757,Z 322.359,A -85,B 0,C 180,E1 -6358.365,E2 -6358.365} C_VEL
LIN {X 0,Y 495.752,Z 322.357,A -85,B 0,C 180,E1 -6359.493,E2 -6359.493} C_VEL
LIN {X 0,Y 495.542,Z 322.733,A -85,B 0,C 180,E1 -6359.941,E2 -6359.941} C_VEL
LIN {X 0,Y 494.638,Z 324.417,A -85,B 0,C 180,E1 -6360.586,E2 -6360.586} C_VEL
LIN {X 0,Y 493.376,Z 327.011,A -85,B 0,C 180,E1 -6361.188,E2 -6361.188} C_VEL
LIN {X 0,Y 491.663,Z 331.423,A -85,B 0,C 180,E1 -6361.97,E2 -6361.97} C_VEL
LIN {X 0,Y 490.729,Z 335.932,A -85,B 0,C 180,E1 -6362.753,E2 -6362.753} C_VEL
LIN {X 0,Y 490.374,Z 344.535,A -85,B 0,C 180,E1 -6364.31,E2 -6364.31} C_VEL
LIN {X 0,Y 493.642,Z 359.74,A -85,B 0,C 180,E1 -6364.698,E2 -6364.698} C_VEL
LIN {X 0,Y 492.622,Z 480.985,A -85,B 0,C 180,E1 -6366.512,E2 -6366.512} C_VEL
LIN {X 0,Y 492.319,Z 495.181,A -85,B 0,C 180,E1 -6366.886,E2 -6366.886} C_VEL
LIN {X 0,Y 491.915,Z 508.998,A -85,B 0,C 180,E1 -6367.421,E2 -6367.421} C_VEL
LIN {X 0,Y 491.42,Z 521.488,A -85,B 0,C 180,E1 -6368.061,E2 -6368.061} C_VEL
LIN {X 0,Y 490.853,Z 534.141,A -85,B 0,C 180,E1 -6368.886,E2 -6368.886} C_VEL
LIN {X 0,Y 490.339,Z 546.346,A -85,B 0,C 180,E1 -6369.88,E2 -6369.88} C_VEL
LIN {X 0,Y 489.869,Z 556.841,A -85,B 0,C 180,E1 -6370.921,E2 -6370.921} C_VEL
LIN {X 0,Y 489.339,Z 566.079,A -85,B 0,C 180,E1 -6372.014,E2 -6372.014} C_VEL
LIN {X 0,Y 488.876,Z 575.074,A -85,B 0,C 180,E1 -6373.291,E2 -6373.291} C_VEL
LIN {X 0,Y 488.564,Z 583.028,A -85,B 0,C 180,E1 -6374.663,E2 -6374.663} C_VEL
LIN {X 0,Y 488.263,Z 590.501,A -85,B 0,C 180,E1 -6376.261,E2 -6376.261} C_VEL
LIN {X 0,Y 488.108,Z 595.179,A -85,B 0,C 180,E1 -6377.528,E2 -6377.528} C_VEL
LIN {X 0,Y 487.98,Z 600.001,A -85,B 0,C 180,E1 -6379.209,E2 -6379.209} C_VEL
LIN {X 0,Y 487.862,Z 603.289,A -85,B 0,C 180,E1 -6380.883,E2 -6380.883} C_VEL
LIN {X 0,Y 487.912,Z 605.147,A -85,B 0,C 180,E1 -6382.552,E2 -6382.552} C_VEL
LIN {X 0,Y 487.934,Z 605.665,A -85,B 0,C 180,E1 -6384.213,E2 -6384.213} C_VEL
LIN {X 0,Y 487.89,Z 604.863,A -85,B 0,C 180,E1 -6385.87,E2 -6385.87} C_VEL
LIN {X 0,Y 487.932,Z 602.733,A -85,B 0,C 180,E1 -6387.523,E2 -6387.523} C_VEL
LIN {X 0,Y 487.905,Z 599.24,A -85,B 0,C 180,E1 -6389.175,E2 -6389.175} C_VEL
LIN {X 0,Y 488.084,Z 595.675,A -85,B 0,C 180,E1 -6390.412,E2 -6390.412} C_VEL
LIN {X 0,Y 488.266,Z 589.475,A -85,B 0,C 180,E1 -6392.062,E2 -6392.062} C_VEL
LIN {X 0,Y 488.428,Z 582.598,A -85,B 0,C 180,E1 -6393.506,E2 -6393.506} C_VEL
LIN {X 0,Y 488.936,Z 575.405,A -85,B 0,C 180,E1 -6394.741,E2 -6394.741} C_VEL
LIN {X 0,Y 489.341,Z 566.8,A -85,B 0,C 180,E1 -6395.977,E2 -6395.977} C_VEL
LIN {X 0,Y 489.839,Z 556.398,A -85,B 0,C 180,E1 -6397.212,E2 -6397.212} C_VEL
LIN {X 0,Y 490.348,Z 544.897,A -85,B 0,C 180,E1 -6398.333,E2 -6398.333} C_VEL
LIN {X 0,Y 490.988,Z 533.113,A -85,B 0,C 180,E1 -6399.267,E2 -6399.267} C_VEL
LIN {X 0,Y 491.506,Z 520.281,A -85,B 0,C 180,E1 -6400.088,E2 -6400.088} C_VEL
LIN {X 0,Y 492.019,Z 506.851,A -85,B 0,C 180,E1 -6400.753,E2 -6400.753} C_VEL
LIN {X 0,Y 492.397,Z 494.438,A -85,B 0,C 180,E1 -6401.213,E2 -6401.213} C_VEL
LIN {X 0,Y 492.655,Z 480.5,A -85,B 0,C 180,E1 -6401.572,E2 -6401.572} C_VEL
LIN {X 0,Y 493.494,Z 359.41,A -85,B 0,C 180,E1 -6403.377,E2 -6403.377} C_VEL
LIN {X 0,Y 490.343,Z 344.392,A -85,B 0,C 180,E1 -6403.756,E2 -6403.756} C_VEL
LIN {X 0,Y 490.631,Z 333.064,A -85,B 0,C 180,E1 -6405.793,E2 -6405.793} C_VEL
LIN {X 0,Y 488.803,Z 323.226,A -85,B 0,C 180,E1 -6407.729,E2 -6407.729} C_VEL
LIN {X 0,Y 488.71,Z 323.234,A -85,B 0,C 180,E1 -6411.07,E2 -6411.07} C_VEL
LIN {X 0,Y 488.683,Z 323.241,A -85,B 0,C 180,E1 -6413.745,E2 -6413.745} C_VEL
LIN {X 0,Y 488.794,Z 323.221,A -85,B 0,C 180,E1 -6416.943,E2 -6416.943} C_VEL
LIN {X 0,Y 488.711,Z 323.232,A -85,B 0,C 180,E1 -6420.362,E2 -6420.362} C_VEL
LIN {X 0,Y 488.736,Z 323.232,A -85,B 0,C 180,E1 -6423.483,E2 -6423.483} C_VEL
LIN {X 0,Y 488.687,Z 323.232,A -85,B 0,C 180,E1 -6426.354,E2 -6426.354} C_VEL
LIN {X 0,Y 488.699,Z 323.236,A -85,B 0,C 180,E1 -6429.253,E2 -6429.253} C_VEL
LIN {X 0,Y 488.704,Z 323.235,A -85,B 0,C 180,E1 -6431.599,E2 -6431.599} C_VEL
LIN {X 0,Y 488.708,Z 323.23,A -85,B 0,C 180,E1 -6434.8,E2 -6434.8} C_VEL
LIN {X 0,Y 488.687,Z 323.237,A -85,B 0,C 180,E1 -6437.473,E2 -6437.473} C_VEL
LIN {X 0,Y 488.728,Z 323.232,A -85,B 0,C 180,E1 -6439.675,E2 -6439.675} C_VEL
LIN {X 0,Y 488.672,Z 323.234,A -85,B 0,C 180,E1 -6442.84,E2 -6442.84} C_VEL
LIN {X 0,Y 488.718,Z 323.228,A -85,B 0,C 180,E1 -6445.886,E2 -6445.886} C_VEL
LIN {X 0,Y 488.683,Z 323.236,A -85,B 0,C 180,E1 -6448.819,E2 -6448.819} C_VEL
LIN {X 0,Y 488.732,Z 323.223,A -85,B 0,C 180,E1 -6451.67,E2 -6451.67} C_VEL
LIN {X 0,Y 488.7,Z 323.23,A -85,B 0,C 180,E1 -6454.441,E2 -6454.441} C_VEL
LIN {X 0,Y 488.71,Z 323.234,A -85,B 0,C 180,E1 -6457.152,E2 -6457.152} C_VEL
LIN {X 0,Y 488.711,Z 323.222,A -85,B 0,C 180,E1 -6459.809,E2 -6459.809} C_VEL
LIN {X 0,Y 488.697,Z 323.232,A -85,B 0,C 180,E1 -6462.422,E2 -6462.422} C_VEL
LIN {X 0,Y 488.745,Z 323.228,A -85,B 0,C 180,E1 -6464.999,E2 -6464.999} C_VEL
LIN {X 0,Y 488.791,Z 323.215,A -85,B 0,C 180,E1 -6468.387,E2 -6468.387} C_VEL
LIN {X 0,Y 488.769,Z 323.222,A -85,B 0,C 180,E1 -6471.732,E2 -6471.732} C_VEL
LIN {X 0,Y 488.82,Z 323.216,A -85,B 0,C 180,E1 -6474.224,E2 -6474.224} C_VEL
LIN {X 0,Y 488.934,Z 323.2,A -85,B 0,C 180,E1 -6477.528,E2 -6477.528} C_VEL
LIN {X 0,Y 488.879,Z 323.211,A -85,B 0,C 180,E1 -6480.823,E2 -6480.823} C_VEL
LIN {X 0,Y 488.924,Z 323.205,A -85,B 0,C 180,E1 -6482.471,E2 -6482.471} C_VEL
LIN {X 0,Y 488.803,Z 323.219,A -85,B 0,C 180,E1 -6485.776,E2 -6485.776} C_VEL
LIN {X 0,Y 488.746,Z 323.231,A -85,B 0,C 180,E1 -6488.267,E2 -6488.267} C_VEL
LIN {X 0,Y 488.79,Z 323.22,A -85,B 0,C 180,E1 -6491.613,E2 -6491.613} C_VEL
LIN {X 0,Y 488.747,Z 323.222,A -85,B 0,C 180,E1 -6495.001,E2 -6495.001} C_VEL
LIN {X 0,Y 488.733,Z 323.231,A -85,B 0,C 180,E1 -6498.443,E2 -6498.443} C_VEL
LIN {X 0,Y 488.694,Z 323.226,A -85,B 0,C 180,E1 -6501.071,E2 -6501.071} C_VEL
LIN {X 0,Y 488.663,Z 323.238,A -85,B 0,C 180,E1 -6503.747,E2 -6503.747} C_VEL
LIN {X 0,Y 488.713,Z 323.228,A -85,B 0,C 180,E1 -6506.928,E2 -6506.928} C_VEL
LIN {X 0,Y 488.713,Z 323.233,A -85,B 0,C 180,E1 -6510.22,E2 -6510.22} C_VEL
LIN {X 0,Y 488.725,Z 323.231,A -85,B 0,C 180,E1 -6513.485,E2 -6513.485} C_VEL
LIN {X 0,Y 488.677,Z 323.236,A -85,B 0,C 180,E1 -6516.356,E2 -6516.356} C_VEL
LIN {X 0,Y 488.692,Z 323.234,A -85,B 0,C 180,E1 -6519.255,E2 -6519.255} C_VEL
LIN {X 0,Y 488.7,Z 323.232,A -85,B 0,C 180,E1 -6521.601,E2 -6521.601} C_VEL
LIN {X 0,Y 488.705,Z 323.23,A -85,B 0,C 180,E1 -6524.802,E2 -6524.802} C_VEL
LIN {X 0,Y 488.685,Z 323.239,A -85,B 0,C 180,E1 -6527.475,E2 -6527.475} C_VEL
LIN {X 0,Y 488.727,Z 323.236,A -85,B 0,C 180,E1 -6529.677,E2 -6529.677} C_VEL
LIN {X 0,Y 488.677,Z 323.238,A -85,B 0,C 180,E1 -6532.842,E2 -6532.842} C_VEL
LIN {X 0,Y 488.73,Z 323.233,A -85,B 0,C 180,E1 -6535.888,E2 -6535.888} C_VEL
LIN {X 0,Y 488.689,Z 323.236,A -85,B 0,C 180,E1 -6538.821,E2 -6538.821} C_VEL
LIN {X 0,Y 488.742,Z 323.232,A -85,B 0,C 180,E1 -6541.672,E2 -6541.672} C_VEL
LIN {X 0,Y 488.789,Z 323.289,A -85,B 0,C 180,E1 -6542.943,E2 -6542.943} C_VEL
LIN {X 0,Y 491.409,Z 335.689,A -85,B 0,C 180,E1 -6545.046,E2 -6545.046} C_VEL
LIN {X 0,Y 491.436,Z 341.715,A -85,B 0,C 180,E1 -6545.993,E2 -6545.993} C_VEL
LIN {X 0,Y 490.688,Z 359.43,A -85,B 0,C 180,E1 -6548.711,E2 -6548.711} C_VEL
LIN {X 0,Y 490.317,Z 369.838,A -85,B 0,C 180,E1 -6550.295,E2 -6550.295} C_VEL
LIN {X 0,Y 493.509,Z 389.263,A -85,B 0,C 180,E1 -6550.716,E2 -6550.716} C_VEL
LIN {X 0,Y 492.485,Z 508.027,A -85,B 0,C 180,E1 -6552.482,E2 -6552.482} C_VEL
LIN {X 0,Y 492.102,Z 522.712,A -85,B 0,C 180,E1 -6552.872,E2 -6552.872} C_VEL
LIN {X 0,Y 491.718,Z 536.042,A -85,B 0,C 180,E1 -6553.391,E2 -6553.391} C_VEL
LIN {X 0,Y 491.167,Z 550.041,A -85,B 0,C 180,E1 -6554.119,E2 -6554.119} C_VEL
LIN {X 0,Y 490.545,Z 562.556,A -85,B 0,C 180,E1 -6554.95,E2 -6554.95} C_VEL
LIN {X 0,Y 490.04,Z 573.995,A -85,B 0,C 180,E1 -6555.889,E2 -6555.889} C_VEL
LIN {X 0,Y 489.51,Z 584.505,A -85,B 0,C 180,E1 -6556.931,E2 -6556.931} C_VEL
LIN {X 0,Y 489.116,Z 593.945,A -85,B 0,C 180,E1 -6558.055,E2 -6558.055} C_VEL
LIN {X 0,Y 488.684,Z 603.586,A -85,B 0,C 180,E1 -6559.435,E2 -6559.435} C_VEL
LIN {X 0,Y 488.337,Z 611.849,A -85,B 0,C 180,E1 -6560.892,E2 -6560.892} C_VEL
LIN {X 0,Y 488.147,Z 617.632,A -85,B 0,C 180,E1 -6562.139,E2 -6562.139} C_VEL
LIN {X 0,Y 488.071,Z 622.765,A -85,B 0,C 180,E1 -6563.498,E2 -6563.498} C_VEL
LIN {X 0,Y 487.96,Z 627.286,A -85,B 0,C 180,E1 -6565.043,E2 -6565.043} C_VEL
LIN {X 0,Y 487.955,Z 630.702,A -85,B 0,C 180,E1 -6566.697,E2 -6566.697} C_VEL
LIN {X 0,Y 487.887,Z 632.72,A -85,B 0,C 180,E1 -6568.349,E2 -6568.349} C_VEL
LIN {X 0,Y 487.817,Z 633.387,A -85,B 0,C 180,E1 -6570,E2 -6570} C_VEL
LIN {X 0,Y 487.887,Z 632.718,A -85,B 0,C 180,E1 -6571.651,E2 -6571.651} C_VEL
LIN {X 0,Y 487.955,Z 630.698,A -85,B 0,C 180,E1 -6573.303,E2 -6573.303} C_VEL
LIN {X 0,Y 487.961,Z 627.277,A -85,B 0,C 180,E1 -6574.957,E2 -6574.957} C_VEL
LIN {X 0,Y 488.04,Z 622.355,A -85,B 0,C 180,E1 -6576.615,E2 -6576.615} C_VEL
LIN {X 0,Y 488.23,Z 615.79,A -85,B 0,C 180,E1 -6578.276,E2 -6578.276} C_VEL
LIN {X 0,Y 488.469,Z 608.485,A -85,B 0,C 180,E1 -6579.733,E2 -6579.733} C_VEL
LIN {X 0,Y 488.881,Z 599.444,A -85,B 0,C 180,E1 -6581.19,E2 -6581.19} C_VEL
LIN {X 0,Y 489.268,Z 589.956,A -85,B 0,C 180,E1 -6582.442,E2 -6582.442} C_VEL
LIN {X 0,Y 489.775,Z 579.463,A -85,B 0,C 180,E1 -6583.59,E2 -6583.59} C_VEL
LIN {X 0,Y 490.305,Z 567.89,A -85,B 0,C 180,E1 -6584.633,E2 -6584.633} C_VEL
LIN {X 0,Y 490.917,Z 555.064,A -85,B 0,C 180,E1 -6585.57,E2 -6585.57} C_VEL
LIN {X 0,Y 491.459,Z 542.553,A -85,B 0,C 180,E1 -6586.298,E2 -6586.298} C_VEL
LIN {X 0,Y 491.894,Z 529.429,A -85,B 0,C 180,E1 -6586.892,E2 -6586.892} C_VEL
LIN {X 0,Y 492.301,Z 516.241,A -85,B 0,C 180,E1 -6587.327,E2 -6587.327} C_VEL
LIN {X 0,Y 492.57,Z 501.119,A -85,B 0,C 180,E1 -6587.649,E2 -6587.649} C_VEL
LIN {X 0,Y 493.491,Z 387.985,A -85,B 0,C 180,E1 -6589.322,E2 -6589.322} C_VEL
LIN {X 0,Y 490.333,Z 369.678,A -85,B 0,C 180,E1 -6589.75,E2 -6589.75} C_VEL
LIN {X 0,Y 491.148,Z 348.955,A -85,B 0,C 180,E1 -6592.949,E2 -6592.949} C_VEL
LIN {X 0,Y 491.659,Z 337.685,A -85,B 0,C 180,E1 -6594.715,E2 -6594.715} C_VEL
LIN {X 0,Y 490.399,Z 330.643,A -85,B 0,C 180,E1 -6595.918,E2 -6595.918} C_VEL
LIN {X 0,Y 488.771,Z 323.228,A -85,B 0,C 180,E1 -6597.261,E2 -6597.261} C_VEL
LIN {X 0,Y 488.707,Z 323.238,A -85,B 0,C 180,E1 -6600.362,E2 -6600.362} C_VEL
LIN {X 0,Y 488.732,Z 323.23,A -85,B 0,C 180,E1 -6603.484,E2 -6603.484} C_VEL
LIN {X 0,Y 488.684,Z 323.238,A -85,B 0,C 180,E1 -6606.355,E2 -6606.355} C_VEL
LIN {X 0,Y 488.695,Z 323.23,A -85,B 0,C 180,E1 -6609.254,E2 -6609.254} C_VEL
LIN {X 0,Y 488.701,Z 323.228,A -85,B 0,C 180,E1 -6611.599,E2 -6611.599} C_VEL
LIN {X 0,Y 488.705,Z 323.229,A -85,B 0,C 180,E1 -6614.801,E2 -6614.801} C_VEL
LIN {X 0,Y 488.684,Z 323.232,A -85,B 0,C 180,E1 -6617.474,E2 -6617.474} C_VEL
LIN {X 0,Y 488.725,Z 323.23,A -85,B 0,C 180,E1 -6619.676,E2 -6619.676} C_VEL
LIN {X 0,Y 488.672,Z 323.235,A -85,B 0,C 180,E1 -6622.841,E2 -6622.841} C_VEL
LIN {X 0,Y 488.722,Z 323.232,A -85,B 0,C 180,E1 -6625.887,E2 -6625.887} C_VEL
LIN {X 0,Y 488.681,Z 323.228,A -85,B 0,C 180,E1 -6628.82,E2 -6628.82} C_VEL
LIN {X 0,Y 488.7,Z 323.228,A -85,B 0,C 180,E1 -6631.669,E2 -6631.669} C_VEL
LIN {X 0,Y 488.698,Z 323.231,A -85,B 0,C 180,E1 -6634.442,E2 -6634.442} C_VEL
LIN {X 0,Y 488.709,Z 323.231,A -85,B 0,C 180,E1 -6637.153,E2 -6637.153} C_VEL
LIN {X 0,Y 488.711,Z 323.234,A -85,B 0,C 180,E1 -6639.81,E2 -6639.81} C_VEL
LIN {X 0,Y 488.695,Z 323.232,A -85,B 0,C 180,E1 -6642.422,E2 -6642.422} C_VEL
LIN {X 0,Y 488.743,Z 323.225,A -85,B 0,C 180,E1 -6644.999,E2 -6644.999} C_VEL
LIN {X 0,Y 488.769,Z 323.219,A -85,B 0,C 180,E1 -6648.387,E2 -6648.387} C_VEL
LIN {X 0,Y 488.739,Z 323.229,A -85,B 0,C 180,E1 -6651.733,E2 -6651.733} C_VEL
LIN {X 0,Y 488.811,Z 323.217,A -85,B 0,C 180,E1 -6654.224,E2 -6654.224} C_VEL
LIN {X 0,Y 488.931,Z 323.205,A -85,B 0,C 180,E1 -6657.529,E2 -6657.529} C_VEL
LIN {X 0,Y 488.924,Z 323.205,A -85,B 0,C 180,E1 -6660,E2 -6660} C_VEL
LIN {X 0,Y 488.936,Z 323.199,A -85,B 0,C 180,E1 -6662.472,E2 -6662.472} C_VEL
LIN {X 0,Y 488.822,Z 323.217,A -85,B 0,C 180,E1 -6665.776,E2 -6665.776} C_VEL
LIN {X 0,Y 488.77,Z 323.22,A -85,B 0,C 180,E1 -6668.268,E2 -6668.268} C_VEL
LIN {X 0,Y 488.791,Z 323.218,A -85,B 0,C 180,E1 -6671.613,E2 -6671.613} C_VEL
LIN {X 0,Y 488.746,Z 323.233,A -85,B 0,C 180,E1 -6675.001,E2 -6675.001} C_VEL
LIN {X 0,Y 488.736,Z 323.228,A -85,B 0,C 180,E1 -6678.443,E2 -6678.443} C_VEL
LIN {X 0,Y 488.696,Z 323.237,A -85,B 0,C 180,E1 -6681.072,E2 -6681.072} C_VEL
LIN {X 0,Y 488.678,Z 323.233,A -85,B 0,C 180,E1 -6683.747,E2 -6683.747} C_VEL
LIN {X 0,Y 488.783,Z 323.226,A -85,B 0,C 180,E1 -6686.944,E2 -6686.944} C_VEL
LIN {X 0,Y 488.701,Z 323.235,A -85,B 0,C 180,E1 -6690.364,E2 -6690.364} C_VEL
LIN {X 0,Y 488.728,Z 323.228,A -85,B 0,C 180,E1 -6693.485,E2 -6693.485} C_VEL
LIN {X 0,Y 488.676,Z 323.239,A -85,B 0,C 180,E1 -6696.356,E2 -6696.356} C_VEL
LIN {X 0,Y 488.696,Z 323.232,A -85,B 0,C 180,E1 -6699.255,E2 -6699.255} C_VEL
LIN {X 0,Y 488.703,Z 323.231,A -85,B 0,C 180,E1 -6701.601,E2 -6701.601} C_VEL
LIN {X 0,Y 488.709,Z 323.235,A -85,B 0,C 180,E1 -6704.803,E2 -6704.803} C_VEL
LIN {X 0,Y 488.689,Z 323.234,A -85,B 0,C 180,E1 -6707.476,E2 -6707.476} C_VEL
LIN {X 0,Y 488.731,Z 323.23,A -85,B 0,C 180,E1 -6709.678,E2 -6709.678} C_VEL
LIN {X 0,Y 488.681,Z 323.236,A -85,B 0,C 180,E1 -6712.842,E2 -6712.842} C_VEL
LIN {X 0,Y 488.735,Z 323.229,A -85,B 0,C 180,E1 -6715.889,E2 -6715.889} C_VEL
LIN {X 0,Y 488.694,Z 323.238,A -85,B 0,C 180,E1 -6718.821,E2 -6718.821} C_VEL
LIN {X 0,Y 488.751,Z 323.331,A -85,B 0,C 180,E1 -6720.289,E2 -6720.289} C_VEL
LIN {X 0,Y 490.53,Z 332.015,A -85,B 0,C 180,E1 -6722.017,E2 -6722.017} C_VEL
LIN {X 0,Y 490.729,Z 335.932,A -85,B 0,C 180,E1 -6722.753,E2 -6722.753} C_VEL
LIN {X 0,Y 489.996,Z 338.359,A -85,B 0,C 180,E1 -6723.14,E2 -6723.14} C_VEL
LIN {X 0,Y 487.355,Z 343.021,A -85,B 0,C 180,E1 -6723.676,E2 -6723.676} C_VEL
LIN {X 0,Y 485.492,Z 347.364,A -85,B 0,C 180,E1 -6724,E2 -6724} C_VEL
LIN {X 0,Y 485.042,Z 351.056,A -85,B 0,C 180,E1 -6724.172,E2 -6724.172} C_VEL
LIN {X 0,Y 485.206,Z 352.336,A -85,B 0,C 180,E1 -6724.21,E2 -6724.21} C_VEL
LIN {X 0,Y 487.01,Z 361.732,A -85,B 0,C 180,E1 -6724.438,E2 -6724.438} C_VEL
LIN {X 0,Y 485.886,Z 481.27,A -85,B 0,C 180,E1 -6726.251,E2 -6726.251} C_VEL
LIN {X 0,Y 485.59,Z 495.434,A -85,B 0,C 180,E1 -6726.632,E2 -6726.632} C_VEL
LIN {X 0,Y 485.122,Z 509.802,A -85,B 0,C 180,E1 -6727.2,E2 -6727.2} C_VEL
LIN {X 0,Y 484.574,Z 523.242,A -85,B 0,C 180,E1 -6727.915,E2 -6727.915} C_VEL
LIN {X 0,Y 483.97,Z 535.094,A -85,B 0,C 180,E1 -6728.714,E2 -6728.714} C_VEL
LIN {X 0,Y 483.439,Z 546.827,A -85,B 0,C 180,E1 -6729.692,E2 -6729.692} C_VEL
LIN {X 0,Y 482.984,Z 556.514,A -85,B 0,C 180,E1 -6730.666,E2 -6730.666} C_VEL
LIN {X 0,Y 482.322,Z 567.279,A -85,B 0,C 180,E1 -6731.963,E2 -6731.963} C_VEL
LIN {X 0,Y 481.849,Z 576.099,A -85,B 0,C 180,E1 -6733.258,E2 -6733.258} C_VEL
LIN {X 0,Y 481.464,Z 584.504,A -85,B 0,C 180,E1 -6734.767,E2 -6734.767} C_VEL
LIN {X 0,Y 481.213,Z 590.326,A -85,B 0,C 180,E1 -6736.056,E2 -6736.056} C_VEL
LIN {X 0,Y 481.067,Z 595.083,A -85,B 0,C 180,E1 -6737.342,E2 -6737.342} C_VEL
LIN {X 0,Y 480.914,Z 599.98,A -85,B 0,C 180,E1 -6739.049,E2 -6739.049} C_VEL
LIN {X 0,Y 480.769,Z 603.35,A -85,B 0,C 180,E1 -6740.747,E2 -6740.747} C_VEL
LIN {X 0,Y 480.823,Z 605.295,A -85,B 0,C 180,E1 -6742.441,E2 -6742.441} C_VEL
LIN {X 0,Y 480.845,Z 605.883,A -85,B 0,C 180,E1 -6744.128,E2 -6744.128} C_VEL
LIN {X 0,Y 480.792,Z 605.148,A -85,B 0,C 180,E1 -6745.809,E2 -6745.809} C_VEL
LIN {X 0,Y 480.843,Z 603.085,A -85,B 0,C 180,E1 -6747.487,E2 -6747.487} C_VEL
LIN {X 0,Y 480.826,Z 599.659,A -85,B 0,C 180,E1 -6749.163,E2 -6749.163} C_VEL
LIN {X 0,Y 481.016,Z 596.163,A -85,B 0,C 180,E1 -6750.419,E2 -6750.419} C_VEL
LIN {X 0,Y 481.203,Z 590.045,A -85,B 0,C 180,E1 -6752.092,E2 -6752.092} C_VEL
LIN {X 0,Y 481.375,Z 583.251,A -85,B 0,C 180,E1 -6753.557,E2 -6753.557} C_VEL
LIN {X 0,Y 481.9,Z 576.146,A -85,B 0,C 180,E1 -6754.81,E2 -6754.81} C_VEL
LIN {X 0,Y 482.349,Z 567.638,A -85,B 0,C 180,E1 -6756.064,E2 -6756.064} C_VEL
LIN {X 0,Y 482.859,Z 557.355,A -85,B 0,C 180,E1 -6757.317,E2 -6757.317} C_VEL
LIN {X 0,Y 483.399,Z 545.989,A -85,B 0,C 180,E1 -6758.454,E2 -6758.454} C_VEL
LIN {X 0,Y 484.045,Z 534.388,A -85,B 0,C 180,E1 -6759.401,E2 -6759.401} C_VEL
LIN {X 0,Y 484.604,Z 521.797,A -85,B 0,C 180,E1 -6760.233,E2 -6760.233} C_VEL
LIN {X 0,Y 485.138,Z 508.754,A -85,B 0,C 180,E1 -6760.908,E2 -6760.908} C_VEL
LIN {X 0,Y 485.534,Z 495.391,A -85,B 0,C 180,E1 -6761.427,E2 -6761.427} C_VEL
LIN {X 0,Y 485.879,Z 480.645,A -85,B 0,C 180,E1 -6761.815,E2 -6761.815} C_VEL
LIN {X 0,Y 486.779,Z 360.546,A -85,B 0,C 180,E1 -6763.628,E2 -6763.628} C_VEL
LIN {X 0,Y 483.452,Z 344.659,A -85,B 0,C 180,E1 -6764.02,E2 -6764.02} C_VEL
LIN {X 0,Y 483.742,Z 334.826,A -85,B 0,C 180,E1 -6765.807,E2 -6765.807} C_VEL
LIN {X 0,Y 481.763,Z 324.103,A -85,B 0,C 180,E1 -6767.926,E2 -6767.926} C_VEL
LIN {X 0,Y 481.706,Z 324.107,A -85,B 0,C 180,E1 -6770.972,E2 -6770.972} C_VEL
LIN {X 0,Y 481.664,Z 324.114,A -85,B 0,C 180,E1 -6774.113,E2 -6774.113} C_VEL
LIN {X 0,Y 481.749,Z 324.1,A -85,B 0,C 180,E1 -6777.138,E2 -6777.138} C_VEL
LIN {X 0,Y 481.68,Z 324.112,A -85,B 0,C 180,E1 -6779.74,E2 -6779.74} C_VEL
LIN {X 0,Y 481.673,Z 324.106,A -85,B 0,C 180,E1 -6782.673,E2 -6782.673} C_VEL
LIN {X 0,Y 481.641,Z 324.113,A -85,B 0,C 180,E1 -6785.708,E2 -6785.708} C_VEL
LIN {X 0,Y 481.669,Z 324.108,A -85,B 0,C 180,E1 -6788.858,E2 -6788.858} C_VEL
LIN {X 0,Y 481.649,Z 324.112,A -85,B 0,C 180,E1 -6791.912,E2 -6791.912} C_VEL
LIN {X 0,Y 481.656,Z 324.107,A -85,B 0,C 180,E1 -6794.456,E2 -6794.456} C_VEL
LIN {X 0,Y 481.643,Z 324.11,A -85,B 0,C 180,E1 -6797.838,E2 -6797.838} C_VEL
LIN {X 0,Y 481.655,Z 324.11,A -85,B 0,C 180,E1 -6800.653,E2 -6800.653} C_VEL
LIN {X 0,Y 481.621,Z 324.12,A -85,B 0,C 180,E1 -6803.375,E2 -6803.375} C_VEL
LIN {X 0,Y 481.67,Z 324.105,A -85,B 0,C 180,E1 -6806.326,E2 -6806.326} C_VEL
LIN {X 0,Y 481.642,Z 324.115,A -85,B 0,C 180,E1 -6809.416,E2 -6809.416} C_VEL
LIN {X 0,Y 481.682,Z 324.099,A -85,B 0,C 180,E1 -6812.166,E2 -6812.166} C_VEL
LIN {X 0,Y 481.668,Z 324.112,A -85,B 0,C 180,E1 -6814.967,E2 -6814.967} C_VEL
LIN {X 0,Y 481.636,Z 324.109,A -85,B 0,C 180,E1 -6817.704,E2 -6817.704} C_VEL
LIN {X 0,Y 481.69,Z 324.098,A -85,B 0,C 180,E1 -6820.392,E2 -6820.392} C_VEL
LIN {X 0,Y 481.662,Z 324.114,A -85,B 0,C 180,E1 -6823.032,E2 -6823.032} C_VEL
LIN {X 0,Y 481.67,Z 324.103,A -85,B 0,C 180,E1 -6825.638,E2 -6825.638} C_VEL
LIN {X 0,Y 481.737,Z 324.092,A -85,B 0,C 180,E1 -6828.214,E2 -6828.214} C_VEL
LIN {X 0,Y 481.724,Z 324.1,A -85,B 0,C 180,E1 -6831.611,E2 -6831.611} C_VEL
LIN {X 0,Y 481.781,Z 324.091,A -85,B 0,C 180,E1 -6834.139,E2 -6834.139} C_VEL
LIN {X 0,Y 481.9,Z 324.076,A -85,B 0,C 180,E1 -6837.492,E2 -6837.492} C_VEL
LIN {X 0,Y 481.832,Z 324.089,A -85,B 0,C 180,E1 -6840.835,E2 -6840.835} C_VEL
LIN {X 0,Y 481.89,Z 324.081,A -85,B 0,C 180,E1 -6842.507,E2 -6842.507} C_VEL
LIN {X 0,Y 481.764,Z 324.096,A -85,B 0,C 180,E1 -6845.861,E2 -6845.861} C_VEL
LIN {X 0,Y 481.705,Z 324.106,A -85,B 0,C 180,E1 -6848.389,E2 -6848.389} C_VEL
LIN {X 0,Y 481.736,Z 324.099,A -85,B 0,C 180,E1 -6851.785,E2 -6851.785} C_VEL
LIN {X 0,Y 481.729,Z 324.095,A -85,B 0,C 180,E1 -6855.224,E2 -6855.224} C_VEL
LIN {X 0,Y 481.694,Z 324.105,A -85,B 0,C 180,E1 -6858.722,E2 -6858.722} C_VEL
LIN {X 0,Y 481.632,Z 324.106,A -85,B 0,C 180,E1 -6861.395,E2 -6861.395} C_VEL
LIN {X 0,Y 481.644,Z 324.116,A -85,B 0,C 180,E1 -6864.115,E2 -6864.115} C_VEL
LIN {X 0,Y 481.682,Z 324.103,A -85,B 0,C 180,E1 -6867.127,E2 -6867.127} C_VEL
LIN {X 0,Y 481.662,Z 324.112,A -85,B 0,C 180,E1 -6869.742,E2 -6869.742} C_VEL
LIN {X 0,Y 481.662,Z 324.108,A -85,B 0,C 180,E1 -6872.675,E2 -6872.675} C_VEL
LIN {X 0,Y 481.631,Z 324.117,A -85,B 0,C 180,E1 -6875.71,E2 -6875.71} C_VEL
LIN {X 0,Y 481.661,Z 324.108,A -85,B 0,C 180,E1 -6878.86,E2 -6878.86} C_VEL
LIN {X 0,Y 481.645,Z 324.112,A -85,B 0,C 180,E1 -6881.914,E2 -6881.914} C_VEL
LIN {X 0,Y 481.652,Z 324.109,A -85,B 0,C 180,E1 -6884.458,E2 -6884.458} C_VEL
LIN {X 0,Y 481.641,Z 324.116,A -85,B 0,C 180,E1 -6887.84,E2 -6887.84} C_VEL
LIN {X 0,Y 481.655,Z 324.111,A -85,B 0,C 180,E1 -6890.655,E2 -6890.655} C_VEL
LIN {X 0,Y 481.626,Z 324.121,A -85,B 0,C 180,E1 -6893.376,E2 -6893.376} C_VEL
LIN {X 0,Y 481.706,Z 324.105,A -85,B 0,C 180,E1 -6896.331,E2 -6896.331} C_VEL
LIN {X 0,Y 481.648,Z 324.117,A -85,B 0,C 180,E1 -6899.418,E2 -6899.418} C_VEL
LIN {X 0,Y 481.708,Z 324.107,A -85,B 0,C 180,E1 -6902.56,E2 -6902.56} C_VEL
LIN {X 0,Y 481.732,Z 324.138,A -85,B 0,C 180,E1 -6902.707,E2 -6902.707} C_VEL
LIN {X 0,Y 484.632,Z 338.253,A -85,B 0,C 180,E1 -6905.131,E2 -6905.131} C_VEL
LIN {X 0,Y 483.938,Z 356.686,A -85,B 0,C 180,E1 -6908.014,E2 -6908.014} C_VEL
LIN {X 0,Y 483.353,Z 369.615,A -85,B 0,C 180,E1 -6910.01,E2 -6910.01} C_VEL
LIN {X 0,Y 486.786,Z 389.866,A -85,B 0,C 180,E1 -6910.462,E2 -6910.462} C_VEL
LIN {X 0,Y 485.7,Z 507.435,A -85,B 0,C 180,E1 -6912.229,E2 -6912.229} C_VEL
LIN {X 0,Y 485.328,Z 522.205,A -85,B 0,C 180,E1 -6912.623,E2 -6912.623} C_VEL
LIN {X 0,Y 484.877,Z 535.672,A -85,B 0,C 180,E1 -6913.149,E2 -6913.149} C_VEL
LIN {X 0,Y 484.292,Z 549.756,A -85,B 0,C 180,E1 -6913.889,E2 -6913.889} C_VEL
LIN {X 0,Y 483.655,Z 562.279,A -85,B 0,C 180,E1 -6914.73,E2 -6914.73} C_VEL
LIN {X 0,Y 483.051,Z 574.922,A -85,B 0,C 180,E1 -6915.788,E2 -6915.788} C_VEL
LIN {X 0,Y 482.456,Z 586.182,A -85,B 0,C 180,E1 -6916.951,E2 -6916.951} C_VEL
LIN {X 0,Y 481.958,Z 596.274,A -85,B 0,C 180,E1 -6918.221,E2 -6918.221} C_VEL
LIN {X 0,Y 481.585,Z 604.651,A -85,B 0,C 180,E1 -6919.49,E2 -6919.49} C_VEL
LIN {X 0,Y 481.257,Z 612.659,A -85,B 0,C 180,E1 -6920.968,E2 -6920.968} C_VEL
LIN {X 0,Y 481.007,Z 619.107,A -85,B 0,C 180,E1 -6922.444,E2 -6922.444} C_VEL
LIN {X 0,Y 480.963,Z 623.015,A -85,B 0,C 180,E1 -6923.535,E2 -6923.535} C_VEL
LIN {X 0,Y 480.891,Z 627.085,A -85,B 0,C 180,E1 -6924.97,E2 -6924.97} C_VEL
LIN {X 0,Y 480.878,Z 630.502,A -85,B 0,C 180,E1 -6926.649,E2 -6926.649} C_VEL
LIN {X 0,Y 480.789,Z 632.519,A -85,B 0,C 180,E1 -6928.325,E2 -6928.325} C_VEL
LIN {X 0,Y 480.741,Z 633.186,A -85,B 0,C 180,E1 -6930,E2 -6930} C_VEL
LIN {X 0,Y 480.789,Z 632.516,A -85,B 0,C 180,E1 -6931.675,E2 -6931.675} C_VEL
LIN {X 0,Y 480.878,Z 630.496,A -85,B 0,C 180,E1 -6933.351,E2 -6933.351} C_VEL
LIN {X 0,Y 480.891,Z 627.074,A -85,B 0,C 180,E1 -6935.03,E2 -6935.03} C_VEL
LIN {X 0,Y 480.959,Z 622.15,A -85,B 0,C 180,E1 -6936.713,E2 -6936.713} C_VEL
LIN {X 0,Y 481.149,Z 615.585,A -85,B 0,C 180,E1 -6938.399,E2 -6938.399} C_VEL
LIN {X 0,Y 481.423,Z 608.284,A -85,B 0,C 180,E1 -6939.877,E2 -6939.877} C_VEL
LIN {X 0,Y 481.876,Z 599.25,A -85,B 0,C 180,E1 -6941.355,E2 -6941.355} C_VEL
LIN {X 0,Y 482.302,Z 589.779,A -85,B 0,C 180,E1 -6942.625,E2 -6942.625} C_VEL
LIN {X 0,Y 482.829,Z 579.302,A -85,B 0,C 180,E1 -6943.789,E2 -6943.789} C_VEL
LIN {X 0,Y 483.388,Z 567.76,A -85,B 0,C 180,E1 -6944.847,E2 -6944.847} C_VEL
LIN {X 0,Y 484.062,Z 554.972,A -85,B 0,C 180,E1 -6945.796,E2 -6945.796} C_VEL
LIN {X 0,Y 484.613,Z 542.941,A -85,B 0,C 180,E1 -6946.511,E2 -6946.511} C_VEL
LIN {X 0,Y 485.103,Z 529.444,A -85,B 0,C 180,E1 -6947.135,E2 -6947.135} C_VEL
LIN {X 0,Y 485.547,Z 516.371,A -85,B 0,C 180,E1 -6947.576,E2 -6947.576} C_VEL
LIN {X 0,Y 485.804,Z 502.999,A -85,B 0,C 180,E1 -6947.876,E2 -6947.876} C_VEL
LIN {X 0,Y 486.849,Z 390.151,A -85,B 0,C 180,E1 -6949.572,E2 -6949.572} C_VEL
LIN {X 0,Y 484.219,Z 373.739,A -85,B 0,C 180,E1 -6949.943,E2 -6949.943} C_VEL
LIN {X 0,Y 483.409,Z 369.523,A -85,B 0,C 180,E1 -6950.053,E2 -6950.053} C_VEL
LIN {X 0,Y 484.266,Z 350.294,A -85,B 0,C 180,E1 -6953.069,E2 -6953.069} C_VEL
LIN {X 0,Y 484.795,Z 339.043,A -85,B 0,C 180,E1 -6954.86,E2 -6954.86} C_VEL
LIN {X 0,Y 482.897,Z 329.2,A -85,B 0,C 180,E1 -6956.585,E2 -6956.585} C_VEL
LIN {X 0,Y 481.71,Z 324.107,A -85,B 0,C 180,E1 -6957.547,E2 -6957.547} C_VEL
LIN {X 0,Y 481.643,Z 324.118,A -85,B 0,C 180,E1 -6960.71,E2 -6960.71} C_VEL
LIN {X 0,Y 481.693,Z 324.107,A -85,B 0,C 180,E1 -6963.732,E2 -6963.732} C_VEL
LIN {X 0,Y 481.624,Z 324.112,A -85,B 0,C 180,E1 -6966.746,E2 -6966.746} C_VEL
LIN {X 0,Y 481.671,Z 324.107,A -85,B 0,C 180,E1 -6969.94,E2 -6969.94} C_VEL
LIN {X 0,Y 481.626,Z 324.11,A -85,B 0,C 180,E1 -6973.146,E2 -6973.146} C_VEL
LIN {X 0,Y 481.651,Z 324.107,A -85,B 0,C 180,E1 -6975.64,E2 -6975.64} C_VEL
LIN {X 0,Y 481.649,Z 324.11,A -85,B 0,C 180,E1 -6978.958,E2 -6978.958} C_VEL
LIN {X 0,Y 481.646,Z 324.117,A -85,B 0,C 180,E1 -6981.992,E2 -6981.992} C_VEL
LIN {X 0,Y 481.681,Z 324.104,A -85,B 0,C 180,E1 -6985.317,E2 -6985.317} C_VEL
LIN {X 0,Y 481.634,Z 324.109,A -85,B 0,C 180,E1 -6988.311,E2 -6988.311} C_VEL
LIN {X 0,Y 481.662,Z 324.1,A -85,B 0,C 180,E1 -6991.216,E2 -6991.216} C_VEL
LIN {X 0,Y 481.654,Z 324.113,A -85,B 0,C 180,E1 -6994.04,E2 -6994.04} C_VEL
LIN {X 0,Y 481.662,Z 324.108,A -85,B 0,C 180,E1 -6996.812,E2 -6996.812} C_VEL
LIN {X 0,Y 481.682,Z 324.108,A -85,B 0,C 180,E1 -6999.502,E2 -6999.502} C_VEL
LIN {X 0,Y 481.675,Z 324.108,A -85,B 0,C 180,E1 -7002.157,E2 -7002.157} C_VEL
LIN {X 0,Y 481.726,Z 324.098,A -85,B 0,C 180,E1 -7004.775,E2 -7004.775} C_VEL
LIN {X 0,Y 481.72,Z 324.098,A -85,B 0,C 180,E1 -7008.215,E2 -7008.215} C_VEL
LIN {X 0,Y 481.697,Z 324.108,A -85,B 0,C 180,E1 -7011.611,E2 -7011.611} C_VEL
LIN {X 0,Y 481.77,Z 324.095,A -85,B 0,C 180,E1 -7014.139,E2 -7014.139} C_VEL
LIN {X 0,Y 481.898,Z 324.081,A -85,B 0,C 180,E1 -7017.493,E2 -7017.493} C_VEL
LIN {X 0,Y 481.894,Z 324.081,A -85,B 0,C 180,E1 -7020,E2 -7020} C_VEL
LIN {X 0,Y 481.902,Z 324.075,A -85,B 0,C 180,E1 -7022.508,E2 -7022.508} C_VEL
LIN {X 0,Y 481.783,Z 324.093,A -85,B 0,C 180,E1 -7025.861,E2 -7025.861} C_VEL
LIN {X 0,Y 481.725,Z 324.098,A -85,B 0,C 180,E1 -7028.389,E2 -7028.389} C_VEL
LIN {X 0,Y 481.737,Z 324.095,A -85,B 0,C 180,E1 -7031.786,E2 -7031.786} C_VEL
LIN {X 0,Y 481.728,Z 324.103,A -85,B 0,C 180,E1 -7035.225,E2 -7035.225} C_VEL
LIN {X 0,Y 481.697,Z 324.108,A -85,B 0,C 180,E1 -7038.723,E2 -7038.723} C_VEL
LIN {X 0,Y 481.635,Z 324.114,A -85,B 0,C 180,E1 -7041.396,E2 -7041.396} C_VEL
LIN {X 0,Y 481.664,Z 324.107,A -85,B 0,C 180,E1 -7044.114,E2 -7044.114} C_VEL
LIN {X 0,Y 481.737,Z 324.101,A -85,B 0,C 180,E1 -7047.14,E2 -7047.14} C_VEL
LIN {X 0,Y 481.67,Z 324.107,A -85,B 0,C 180,E1 -7049.742,E2 -7049.742} C_VEL
LIN {X 0,Y 481.665,Z 324.114,A -85,B 0,C 180,E1 -7052.675,E2 -7052.675} C_VEL
LIN {X 0,Y 481.631,Z 324.112,A -85,B 0,C 180,E1 -7055.711,E2 -7055.711} C_VEL
LIN {X 0,Y 481.665,Z 324.111,A -85,B 0,C 180,E1 -7058.86,E2 -7058.86} C_VEL
LIN {X 0,Y 481.648,Z 324.112,A -85,B 0,C 180,E1 -7061.914,E2 -7061.914} C_VEL
LIN {X 0,Y 481.656,Z 324.115,A -85,B 0,C 180,E1 -7064.458,E2 -7064.458} C_VEL
LIN {X 0,Y 481.645,Z 324.113,A -85,B 0,C 180,E1 -7067.84,E2 -7067.84} C_VEL
LIN {X 0,Y 481.679,Z 324.112,A -85,B 0,C 180,E1 -7070.652,E2 -7070.652} C_VEL
LIN {X 0,Y 481.63,Z 324.113,A -85,B 0,C 180,E1 -7073.377,E2 -7073.377} C_VEL
LIN {X 0,Y 481.71,Z 324.11,A -85,B 0,C 180,E1 -7076.331,E2 -7076.331} C_VEL
LIN {X 0,Y 481.716,Z 324.167,A -85,B 0,C 180,E1 -7080.021,E2 -7080.021} C_VEL
LIN {X 0,Y 483.748,Z 334.263,A -85,B 0,C 180,E1 -7082.062,E2 -7082.062} C_VEL
LIN {X 0,Y 483.673,Z 341.903,A -85,B 0,C 180,E1 -7083.485,E2 -7083.485} C_VEL
LIN {X 0,Y 483.548,Z 344.795,A -85,B 0,C 180,E1 -7084.014,E2 -7084.014} C_VEL
LIN {X 0,Y 485.206,Z 352.336,A -85,B 0,C 180,E1 -7084.21,E2 -7084.21} C_VEL
LIN {X 0,Y 485.581,Z 356.182,A -85,B 0,C 180,E1 -7084.287,E2 -7084.287} C_VEL
LIN {X 0,Y 485.295,Z 360.084,A -85,B 0,C 180,E1 -7084.335,E2 -7084.335} C_VEL
LIN {X 0,Y 483.524,Z 367.84,A -85,B 0,C 180,E1 -7084.375,E2 -7084.375} C_VEL
LIN {X 0,Y 481.316,Z 375.661,A -85,B 0,C 180,E1 -7084.397,E2 -7084.397} C_VEL
LIN {X 0,Y 480.281,Z 381.607,A -85,B 0,C 180,E1 -7084.443,E2 -7084.443} C_VEL
LIN {X 0,Y 480.181,Z 383.607,A -85,B 0,C 180,E1 -7084.47,E2 -7084.47} C_VEL
LIN {X 0,Y 479.177,Z 481.718,A -85,B 0,C 180,E1 -7085.984,E2 -7085.984} C_VEL
LIN {X 0,Y 478.848,Z 495.777,A -85,B 0,C 180,E1 -7086.369,E2 -7086.369} C_VEL
LIN {X 0,Y 478.384,Z 509.526,A -85,B 0,C 180,E1 -7086.917,E2 -7086.917} C_VEL
LIN {X 0,Y 477.812,Z 522.353,A -85,B 0,C 180,E1 -7087.598,E2 -7087.598} C_VEL
LIN {X 0,Y 477.211,Z 534.258,A -85,B 0,C 180,E1 -7088.397,E2 -7088.397} C_VEL
LIN {X 0,Y 476.625,Z 546.162,A -85,B 0,C 180,E1 -7089.388,E2 -7089.388} C_VEL
LIN {X 0,Y 476.078,Z 556.212,A -85,B 0,C 180,E1 -7090.399,E2 -7090.399} C_VEL
LIN {X 0,Y 475.411,Z 566.869,A -85,B 0,C 180,E1 -7091.692,E2 -7091.692} C_VEL
LIN {X 0,Y 474.896,Z 575.783,A -85,B 0,C 180,E1 -7093.006,E2 -7093.006} C_VEL
LIN {X 0,Y 474.574,Z 582.955,A -85,B 0,C 180,E1 -7094.28,E2 -7094.28} C_VEL
LIN {X 0,Y 474.192,Z 590.176,A -85,B 0,C 180,E1 -7095.845,E2 -7095.845} C_VEL
LIN {X 0,Y 474.028,Z 595.004,A -85,B 0,C 180,E1 -7097.151,E2 -7097.151} C_VEL
LIN {X 0,Y 473.859,Z 599.97,A -85,B 0,C 180,E1 -7098.884,E2 -7098.884} C_VEL
LIN {X 0,Y 473.678,Z 603.406,A -85,B 0,C 180,E1 -7100.607,E2 -7100.607} C_VEL
LIN {X 0,Y 473.733,Z 605.427,A -85,B 0,C 180,E1 -7102.327,E2 -7102.327} C_VEL
LIN {X 0,Y 473.759,Z 606.093,A -85,B 0,C 180,E1 -7104.04,E2 -7104.04} C_VEL
LIN {X 0,Y 473.698,Z 605.429,A -85,B 0,C 180,E1 -7105.746,E2 -7105.746} C_VEL
LIN {X 0,Y 473.797,Z 604.594,A -85,B 0,C 180,E1 -7106.599,E2 -7106.599} C_VEL
LIN {X 0,Y 473.767,Z 601.924,A -85,B 0,C 180,E1 -7108.3,E2 -7108.3} C_VEL
LIN {X 0,Y 473.786,Z 597.849,A -85,B 0,C 180,E1 -7110,E2 -7110} C_VEL
LIN {X 0,Y 474.017,Z 593.824,A -85,B 0,C 180,E1 -7111.274,E2 -7111.274} C_VEL
LIN {X 0,Y 474.075,Z 588.817,A -85,B 0,C 180,E1 -7112.549,E2 -7112.549} C_VEL
LIN {X 0,Y 474.587,Z 581.658,A -85,B 0,C 180,E1 -7114.033,E2 -7114.033} C_VEL
LIN {X 0,Y 475.055,Z 572.843,A -85,B 0,C 180,E1 -7115.518,E2 -7115.518} C_VEL
LIN {X 0,Y 475.638,Z 563.598,A -85,B 0,C 180,E1 -7116.788,E2 -7116.788} C_VEL
LIN {X 0,Y 476.18,Z 553.478,A -85,B 0,C 180,E1 -7117.945,E2 -7117.945} C_VEL
LIN {X 0,Y 476.691,Z 542.861,A -85,B 0,C 180,E1 -7118.955,E2 -7118.955} C_VEL
LIN {X 0,Y 477.35,Z 531.327,A -85,B 0,C 180,E1 -7119.855,E2 -7119.855} C_VEL
LIN {X 0,Y 477.881,Z 519.734,A -85,B 0,C 180,E1 -7120.593,E2 -7120.593} C_VEL
LIN {X 0,Y 478.42,Z 505.889,A -85,B 0,C 180,E1 -7121.277,E2 -7121.277} C_VEL
LIN {X 0,Y 478.906,Z 492.93,A -85,B 0,C 180,E1 -7121.748,E2 -7121.748} C_VEL
LIN {X 0,Y 479.1,Z 479.136,A -85,B 0,C 180,E1 -7122.092,E2 -7122.092} C_VEL
LIN {X 0,Y 480.131,Z 361.919,A -85,B 0,C 180,E1 -7123.876,E2 -7123.876} C_VEL
LIN {X 0,Y 476.546,Z 344.861,A -85,B 0,C 180,E1 -7124.302,E2 -7124.302} C_VEL
LIN {X 0,Y 476.831,Z 336.585,A -85,B 0,C 180,E1 -7125.823,E2 -7125.823} C_VEL
LIN {X 0,Y 474.942,Z 326.185,A -85,B 0,C 180,E1 -7127.881,E2 -7127.881} C_VEL
LIN {X 0,Y 474.693,Z 324.984,A -85,B 0,C 180,E1 -7128.178,E2 -7128.178} C_VEL
LIN {X 0,Y 474.638,Z 324.988,A -85,B 0,C 180,E1 -7131.116,E2 -7131.116} C_VEL
LIN {X 0,Y 474.643,Z 324.985,A -85,B 0,C 180,E1 -7134.493,E2 -7134.493} C_VEL
LIN {X 0,Y 474.683,Z 324.981,A -85,B 0,C 180,E1 -7137.333,E2 -7137.333} C_VEL
LIN {X 0,Y 474.605,Z 324.988,A -85,B 0,C 180,E1 -7140.809,E2 -7140.809} C_VEL
LIN {X 0,Y 474.638,Z 324.986,A -85,B 0,C 180,E1 -7143.983,E2 -7143.983} C_VEL
LIN {X 0,Y 474.573,Z 324.991,A -85,B 0,C 180,E1 -7146.899,E2 -7146.899} C_VEL
LIN {X 0,Y 474.626,Z 324.983,A -85,B 0,C 180,E1 -7149.646,E2 -7149.646} C_VEL
LIN {X 0,Y 474.612,Z 324.988,A -85,B 0,C 180,E1 -7152.933,E2 -7152.933} C_VEL
LIN {X 0,Y 474.605,Z 324.989,A -85,B 0,C 180,E1 -7155.894,E2 -7155.894} C_VEL
LIN {X 0,Y 474.622,Z 324.986,A -85,B 0,C 180,E1 -7159.04,E2 -7159.04} C_VEL
LIN {X 0,Y 474.603,Z 324.987,A -85,B 0,C 180,E1 -7161.703,E2 -7161.703} C_VEL
LIN {X 0,Y 474.616,Z 324.988,A -85,B 0,C 180,E1 -7164.724,E2 -7164.724} C_VEL
LIN {X 0,Y 474.627,Z 324.985,A -85,B 0,C 180,E1 -7167.787,E2 -7167.787} C_VEL
LIN {X 0,Y 474.614,Z 324.99,A -85,B 0,C 180,E1 -7170.884,E2 -7170.884} C_VEL
LIN {X 0,Y 474.619,Z 324.984,A -85,B 0,C 180,E1 -7173.625,E2 -7173.625} C_VEL
LIN {X 0,Y 474.624,Z 324.988,A -85,B 0,C 180,E1 -7176.641,E2 -7176.641} C_VEL
LIN {X 0,Y 474.641,Z 324.974,A -85,B 0,C 180,E1 -7180.089,E2 -7180.089} C_VEL
LIN {X 0,Y 474.622,Z 324.99,A -85,B 0,C 180,E1 -7182.773,E2 -7182.773} C_VEL
LIN {X 0,Y 474.629,Z 324.981,A -85,B 0,C 180,E1 -7185.42,E2 -7185.42} C_VEL
LIN {X 0,Y 474.691,Z 324.968,A -85,B 0,C 180,E1 -7188.037,E2 -7188.037} C_VEL
LIN {X 0,Y 474.696,Z 324.976,A -85,B 0,C 180,E1 -7191.486,E2 -7191.486} C_VEL
LIN {X 0,Y 474.745,Z 324.967,A -85,B 0,C 180,E1 -7194.052,E2 -7194.052} C_VEL
LIN {X 0,Y 474.867,Z 324.952,A -85,B 0,C 180,E1 -7197.455,E2 -7197.455} C_VEL
LIN {X 0,Y 474.862,Z 324.957,A -85,B 0,C 180,E1 -7200,E2 -7200} C_VEL
LIN {X 0,Y 474.855,Z 324.956,A -85,B 0,C 180,E1 -7202.545,E2 -7202.545} C_VEL
LIN {X 0,Y 474.726,Z 324.974,A -85,B 0,C 180,E1 -7205.948,E2 -7205.948} C_VEL
LIN {X 0,Y 474.681,Z 324.978,A -85,B 0,C 180,E1 -7208.514,E2 -7208.514} C_VEL
LIN {X 0,Y 474.69,Z 324.979,A -85,B 0,C 180,E1 -7211.963,E2 -7211.963} C_VEL
LIN {X 0,Y 474.686,Z 324.972,A -85,B 0,C 180,E1 -7215.456,E2 -7215.456} C_VEL
LIN {X 0,Y 474.649,Z 324.981,A -85,B 0,C 180,E1 -7219.011,E2 -7219.011} C_VEL
LIN {X 0,Y 474.575,Z 324.987,A -85,B 0,C 180,E1 -7221.729,E2 -7221.729} C_VEL
LIN {X 0,Y 474.624,Z 324.985,A -85,B 0,C 180,E1 -7224.495,E2 -7224.495} C_VEL
LIN {X 0,Y 474.626,Z 324.983,A -85,B 0,C 180,E1 -7227.324,E2 -7227.324} C_VEL
LIN {X 0,Y 474.592,Z 324.991,A -85,B 0,C 180,E1 -7230.231,E2 -7230.231} C_VEL
LIN {X 0,Y 474.633,Z 324.984,A -85,B 0,C 180,E1 -7233.221,E2 -7233.221} C_VEL
LIN {X 0,Y 474.582,Z 324.992,A -85,B 0,C 180,E1 -7236.324,E2 -7236.324} C_VEL
LIN {X 0,Y 474.619,Z 324.992,A -85,B 0,C 180,E1 -7239.648,E2 -7239.648} C_VEL
LIN {X 0,Y 474.607,Z 324.986,A -85,B 0,C 180,E1 -7242.935,E2 -7242.935} C_VEL
LIN {X 0,Y 474.602,Z 324.993,A -85,B 0,C 180,E1 -7245.896,E2 -7245.896} C_VEL
LIN {X 0,Y 474.622,Z 324.987,A -85,B 0,C 180,E1 -7249.042,E2 -7249.042} C_VEL
LIN {X 0,Y 474.605,Z 324.996,A -85,B 0,C 180,E1 -7251.705,E2 -7251.705} C_VEL
LIN {X 0,Y 474.625,Z 324.989,A -85,B 0,C 180,E1 -7254.727,E2 -7254.727} C_VEL
LIN {X 0,Y 474.632,Z 324.989,A -85,B 0,C 180,E1 -7257.789,E2 -7257.789} C_VEL
LIN {X 0,Y 474.621,Z 324.99,A -85,B 0,C 180,E1 -7260.885,E2 -7260.885} C_VEL
LIN {X 0,Y 474.682,Z 325.131,A -85,B 0,C 180,E1 -7262.492,E2 -7262.492} C_VEL
LIN {X 0,Y 477.689,Z 339.361,A -85,B 0,C 180,E1 -7264.978,E2 -7264.978} C_VEL
LIN {X 0,Y 477.193,Z 352.252,A -85,B 0,C 180,E1 -7267.028,E2 -7267.028} C_VEL
LIN {X 0,Y 476.416,Z 369.435,A -85,B 0,C 180,E1 -7269.728,E2 -7269.728} C_VEL
LIN {X 0,Y 480.042,Z 390.839,A -85,B 0,C 180,E1 -7270.21,E2 -7270.21} C_VEL
LIN {X 0,Y 478.896,Z 507.846,A -85,B 0,C 180,E1 -7271.996,E2 -7271.996} C_VEL
LIN {X 0,Y 478.512,Z 522.561,A -85,B 0,C 180,E1 -7272.4,E2 -7272.4} C_VEL
LIN {X 0,Y 477.987,Z 536.721,A -85,B 0,C 180,E1 -7272.972,E2 -7272.972} C_VEL
LIN {X 0,Y 477.446,Z 549.48,A -85,B 0,C 180,E1 -7273.659,E2 -7273.659} C_VEL
LIN {X 0,Y 476.796,Z 561.933,A -85,B 0,C 180,E1 -7274.505,E2 -7274.505} C_VEL
LIN {X 0,Y 476.147,Z 573.432,A -85,B 0,C 180,E1 -7275.468,E2 -7275.468} C_VEL
LIN {X 0,Y 475.562,Z 583.989,A -85,B 0,C 180,E1 -7276.541,E2 -7276.541} C_VEL
LIN {X 0,Y 475.079,Z 594.51,A -85,B 0,C 180,E1 -7277.835,E2 -7277.835} C_VEL
LIN {X 0,Y 474.632,Z 603.136,A -85,B 0,C 180,E1 -7279.118,E2 -7279.118} C_VEL
LIN {X 0,Y 474.264,Z 611.422,A -85,B 0,C 180,E1 -7280.619,E2 -7280.619} C_VEL
LIN {X 0,Y 474.022,Z 617.213,A -85,B 0,C 180,E1 -7281.903,E2 -7281.903} C_VEL
LIN {X 0,Y 473.869,Z 623.195,A -85,B 0,C 180,E1 -7283.557,E2 -7283.557} C_VEL
LIN {X 0,Y 473.821,Z 626.881,A -85,B 0,C 180,E1 -7284.894,E2 -7284.894} C_VEL
LIN {X 0,Y 473.785,Z 630.299,A -85,B 0,C 180,E1 -7286.598,E2 -7286.598} C_VEL
LIN {X 0,Y 473.695,Z 632.317,A -85,B 0,C 180,E1 -7288.3,E2 -7288.3} C_VEL
LIN {X 0,Y 473.667,Z 632.985,A -85,B 0,C 180,E1 -7290,E2 -7290} C_VEL
LIN {X 0,Y 473.695,Z 632.315,A -85,B 0,C 180,E1 -7291.7,E2 -7291.7} C_VEL
LIN {X 0,Y 473.785,Z 630.295,A -85,B 0,C 180,E1 -7293.402,E2 -7293.402} C_VEL
LIN {X 0,Y 473.822,Z 626.876,A -85,B 0,C 180,E1 -7295.106,E2 -7295.106} C_VEL
LIN {X 0,Y 473.889,Z 621.957,A -85,B 0,C 180,E1 -7296.814,E2 -7296.814} C_VEL
LIN {X 0,Y 474.084,Z 615.399,A -85,B 0,C 180,E1 -7298.525,E2 -7298.525} C_VEL
LIN {X 0,Y 474.358,Z 608.109,A -85,B 0,C 180,E1 -7300.025,E2 -7300.025} C_VEL
LIN {X 0,Y 474.872,Z 599.098,A -85,B 0,C 180,E1 -7301.525,E2 -7301.525} C_VEL
LIN {X 0,Y 475.31,Z 589.646,A -85,B 0,C 180,E1 -7302.814,E2 -7302.814} C_VEL
LIN {X 0,Y 475.882,Z 579.2,A -85,B 0,C 180,E1 -7303.994,E2 -7303.994} C_VEL
LIN {X 0,Y 476.502,Z 567.69,A -85,B 0,C 180,E1 -7305.067,E2 -7305.067} C_VEL
LIN {X 0,Y 477.22,Z 554.942,A -85,B 0,C 180,E1 -7306.029,E2 -7306.029} C_VEL
LIN {X 0,Y 477.9,Z 541.668,A -85,B 0,C 180,E1 -7306.822,E2 -7306.822} C_VEL
LIN {X 0,Y 478.349,Z 528.396,A -85,B 0,C 180,E1 -7307.435,E2 -7307.435} C_VEL
LIN {X 0,Y 478.876,Z 514.123,A -85,B 0,C 180,E1 -7307.905,E2 -7307.905} C_VEL
LIN {X 0,Y 479.204,Z 498.799,A -85,B 0,C 180,E1 -7308.214,E2 -7308.214} C_VEL
LIN {X 0,Y 480.166,Z 389.999,A -85,B 0,C 180,E1 -7309.872,E2 -7309.872} C_VEL
LIN {X 0,Y 476.529,Z 369.328,A -85,B 0,C 180,E1 -7310.372,E2 -7310.372} C_VEL
LIN {X 0,Y 477.387,Z 351.645,A -85,B 0,C 180,E1 -7313.191,E2 -7313.191} C_VEL
LIN {X 0,Y 477.924,Z 340.409,A -85,B 0,C 180,E1 -7315.009,E2 -7315.009} C_VEL
LIN {X 0,Y 475.335,Z 327.783,A -85,B 0,C 180,E1 -7317.28,E2 -7317.28} C_VEL
LIN {X 0,Y 474.676,Z 324.984,A -85,B 0,C 180,E1 -7317.829,E2 -7317.829} C_VEL
LIN {X 0,Y 474.595,Z 324.993,A -85,B 0,C 180,E1 -7321.217,E2 -7321.217} C_VEL
LIN {X 0,Y 474.63,Z 324.99,A -85,B 0,C 180,E1 -7324.24,E2 -7324.24} C_VEL
LIN {X 0,Y 474.587,Z 324.984,A -85,B 0,C 180,E1 -7327.383,E2 -7327.383} C_VEL
LIN {X 0,Y 474.622,Z 324.983,A -85,B 0,C 180,E1 -7329.647,E2 -7329.647} C_VEL
LIN {X 0,Y 474.6,Z 324.986,A -85,B 0,C 180,E1 -7332.934,E2 -7332.934} C_VEL
LIN {X 0,Y 474.602,Z 324.987,A -85,B 0,C 180,E1 -7335.894,E2 -7335.894} C_VEL
LIN {X 0,Y 474.62,Z 324.985,A -85,B 0,C 180,E1 -7339.04,E2 -7339.04} C_VEL
LIN {X 0,Y 474.601,Z 324.991,A -85,B 0,C 180,E1 -7341.703,E2 -7341.703} C_VEL
LIN {X 0,Y 474.618,Z 324.985,A -85,B 0,C 180,E1 -7344.725,E2 -7344.725} C_VEL
LIN {X 0,Y 474.625,Z 324.99,A -85,B 0,C 180,E1 -7347.787,E2 -7347.787} C_VEL
LIN {X 0,Y 474.595,Z 324.98,A -85,B 0,C 180,E1 -7350.888,E2 -7350.888} C_VEL
LIN {X 0,Y 474.603,Z 324.991,A -85,B 0,C 180,E1 -7353.625,E2 -7353.625} C_VEL
LIN {X 0,Y 474.623,Z 324.985,A -85,B 0,C 180,E1 -7356.641,E2 -7356.641} C_VEL
LIN {X 0,Y 474.64,Z 324.986,A -85,B 0,C 180,E1 -7360.089,E2 -7360.089} C_VEL
LIN {X 0,Y 474.621,Z 324.984,A -85,B 0,C 180,E1 -7362.774,E2 -7362.774} C_VEL
LIN {X 0,Y 474.627,Z 324.988,A -85,B 0,C 180,E1 -7365.421,E2 -7365.421} C_VEL
LIN {X 0,Y 474.678,Z 324.977,A -85,B 0,C 180,E1 -7368.037,E2 -7368.037} C_VEL
LIN {X 0,Y 474.646,Z 324.989,A -85,B 0,C 180,E1 -7371.485,E2 -7371.485} C_VEL
LIN {X 0,Y 474.732,Z 324.972,A -85,B 0,C 180,E1 -7374.052,E2 -7374.052} C_VEL
LIN {X 0,Y 474.863,Z 324.957,A -85,B 0,C 180,E1 -7377.455,E2 -7377.455} C_VEL
LIN {X 0,Y 474.863,Z 324.956,A -85,B 0,C 180,E1 -7380,E2 -7380} C_VEL
LIN {X 0,Y 474.869,Z 324.951,A -85,B 0,C 180,E1 -7382.545,E2 -7382.545} C_VEL
LIN {X 0,Y 474.747,Z 324.969,A -85,B 0,C 180,E1 -7385.948,E2 -7385.948} C_VEL
LIN {X 0,Y 474.697,Z 324.974,A -85,B 0,C 180,E1 -7388.514,E2 -7388.514} C_VEL
LIN {X 0,Y 474.691,Z 324.972,A -85,B 0,C 180,E1 -7391.963,E2 -7391.963} C_VEL
LIN {X 0,Y 474.687,Z 324.977,A -85,B 0,C 180,E1 -7395.456,E2 -7395.456} C_VEL
LIN {X 0,Y 474.652,Z 324.988,A -85,B 0,C 180,E1 -7399.011,E2 -7399.011} C_VEL
LIN {X 0,Y 474.578,Z 324.991,A -85,B 0,C 180,E1 -7401.73,E2 -7401.73} C_VEL
LIN {X 0,Y 474.647,Z 324.984,A -85,B 0,C 180,E1 -7404.494,E2 -7404.494} C_VEL
LIN {X 0,Y 474.672,Z 324.979,A -85,B 0,C 180,E1 -7407.335,E2 -7407.335} C_VEL
LIN {X 0,Y 474.597,Z 324.992,A -85,B 0,C 180,E1 -7410.811,E2 -7410.811} C_VEL
LIN {X 0,Y 474.631,Z 324.984,A -85,B 0,C 180,E1 -7413.985,E2 -7413.985} C_VEL
LIN {X 0,Y 474.565,Z 324.994,A -85,B 0,C 180,E1 -7416.9,E2 -7416.9} C_VEL
LIN {X 0,Y 474.613,Z 324.985,A -85,B 0,C 180,E1 -7419.647,E2 -7419.647} C_VEL
LIN {X 0,Y 474.611,Z 324.99,A -85,B 0,C 180,E1 -7422.935,E2 -7422.935} C_VEL
LIN {X 0,Y 474.606,Z 324.99,A -85,B 0,C 180,E1 -7425.896,E2 -7425.896} C_VEL
LIN {X 0,Y 474.625,Z 324.987,A -85,B 0,C 180,E1 -7429.042,E2 -7429.042} C_VEL
LIN {X 0,Y 474.609,Z 324.99,A -85,B 0,C 180,E1 -7431.705,E2 -7431.705} C_VEL
LIN {X 0,Y 474.629,Z 324.985,A -85,B 0,C 180,E1 -7434.727,E2 -7434.727} C_VEL
LIN {X 0,Y 474.637,Z 324.99,A -85,B 0,C 180,E1 -7437.789,E2 -7437.789} C_VEL
LIN {X 0,Y 474.678,Z 325.162,A -85,B 0,C 180,E1 -7439.776,E2 -7439.776} C_VEL
LIN {X 0,Y 476.784,Z 335.27,A -85,B 0,C 180,E1 -7441.857,E2 -7441.857} C_VEL
LIN {X 0,Y 476.901,Z 340.285,A -85,B 0,C 180,E1 -7442.817,E2 -7442.817} C_VEL
LIN {X 0,Y 476.689,Z 344.98,A -85,B 0,C 180,E1 -7443.691,E2 -7443.691} C_VEL
LIN {X 0,Y 480.383,Z 362.724,A -85,B 0,C 180,E1 -7444.151,E2 -7444.151} C_VEL
LIN {X 0,Y 480.181,Z 383.607,A -85,B 0,C 180,E1 -7444.47,E2 -7444.47} C_VEL
LIN {X 0,Y 479.517,Z 389.453,A -85,B 0,C 180,E1 -7444.531,E2 -7444.531} C_VEL
LIN {X 0,Y 474.005,Z 408.501,A -85,B 0,C 180,E1 -7444.579,E2 -7444.579} C_VEL
LIN {X 0,Y 473.269,Z 414.35,A -85,B 0,C 180,E1 -7444.639,E2 -7444.639} C_VEL
LIN {X 0,Y 472.472,Z 482.277,A -85,B 0,C 180,E1 -7445.709,E2 -7445.709} C_VEL
LIN {X 0,Y 472.125,Z 496.995,A -85,B 0,C 180,E1 -7446.128,E2 -7446.128} C_VEL
LIN {X 0,Y 471.566,Z 511.616,A -85,B 0,C 180,E1 -7446.738,E2 -7446.738} C_VEL
LIN {X 0,Y 470.984,Z 524.492,A -85,B 0,C 180,E1 -7447.458,E2 -7447.458} C_VEL
LIN {X 0,Y 470.27,Z 536.36,A -85,B 0,C 180,E1 -7448.292,E2 -7448.292} C_VEL
LIN {X 0,Y 469.662,Z 547.921,A -85,B 0,C 180,E1 -7449.298,E2 -7449.298} C_VEL
LIN {X 0,Y 469.128,Z 557.503,A -85,B 0,C 180,E1 -7450.302,E2 -7450.302} C_VEL
LIN {X 0,Y 468.512,Z 566.683,A -85,B 0,C 180,E1 -7451.439,E2 -7451.439} C_VEL
LIN {X 0,Y 467.938,Z 575.496,A -85,B 0,C 180,E1 -7452.745,E2 -7452.745} C_VEL
LIN {X 0,Y 467.494,Z 584.082,A -85,B 0,C 180,E1 -7454.3,E2 -7454.3} C_VEL
LIN {X 0,Y 467.189,Z 590.045,A -85,B 0,C 180,E1 -7455.629,E2 -7455.629} C_VEL
LIN {X 0,Y 466.978,Z 594.943,A -85,B 0,C 180,E1 -7456.953,E2 -7456.953} C_VEL
LIN {X 0,Y 466.792,Z 599.973,A -85,B 0,C 180,E1 -7458.713,E2 -7458.713} C_VEL
LIN {X 0,Y 466.589,Z 603.472,A -85,B 0,C 180,E1 -7460.463,E2 -7460.463} C_VEL
LIN {X 0,Y 466.637,Z 605.553,A -85,B 0,C 180,E1 -7462.21,E2 -7462.21} C_VEL
LIN {X 0,Y 466.669,Z 606.286,A -85,B 0,C 180,E1 -7463.949,E2 -7463.949} C_VEL
LIN {X 0,Y 466.61,Z 605.694,A -85,B 0,C 180,E1 -7465.681,E2 -7465.681} C_VEL
LIN {X 0,Y 466.704,Z 604.896,A -85,B 0,C 180,E1 -7466.547,E2 -7466.547} C_VEL
LIN {X 0,Y 466.685,Z 602.291,A -85,B 0,C 180,E1 -7468.274,E2 -7468.274} C_VEL
